KUKA KRL program: MyProgram_334().src

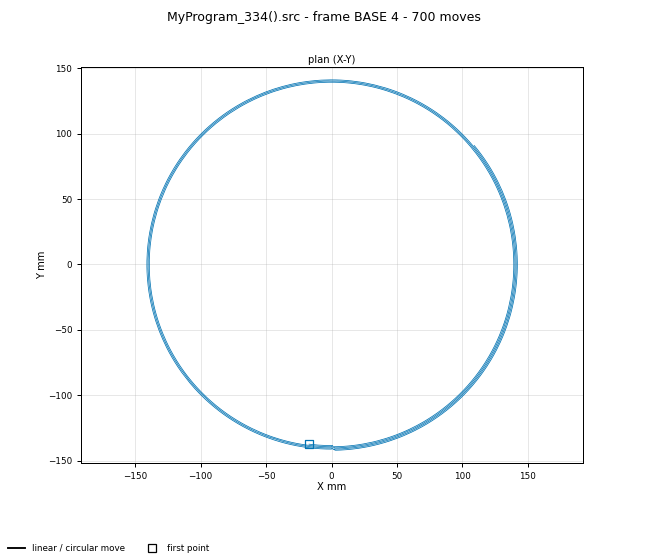
[picture p0: tool path of MyProgram_334().src in frame BASE 4, 700 of 700 moves have a stored position in this frame; points joined in program order, loops and branches not executed]
&ACCESS RVP
&REL 1
&PARAM TEMPLATE = C:\KRC\Roboter\Template\vorgabe
&PARAM EDITMASK = *
DEF MyProgram_334()
; ---- Setting reference (Base) ----
$BASE = BASE_DATA[4]

; --------------------------
; ---- Setting tool (TCP) ----
$TOOL = TOOL_DATA[3]
; --------------------------

$VEL.CP = VEL_APROX_PRINT
Startdeposition()
$VEL.CP = VEL_PRINT
LIN {X -17.1931,Y -137.3704,Z 189,A -88.3722,B 1.6874,C 0.25,E1 1.6941,E2 181.411} C_DIS
LIN {X -13.4645,Y -137.7837,Z 189,A -87.0235,B 1.6872,C 0.2509,E1 1.6978,E2 180.0902} C_DIS
LIN {X -10.3539,Y -138.0524,Z 189,A -85.5339,B 1.6873,C 0.25,E1 1.7021,E2 178.5723} C_DIS
LIN {X -7.0478,Y -138.2604,Z 189,A -84.1441,B 1.6873,C 0.2498,E1 1.706,E2 177.1792} C_DIS
LIN {X -4.0759,Y -138.3801,Z 189,A -82.9485,B 1.6873,C 0.2498,E1 1.7093,E2 175.9881} C_DIS
LIN {X 0.9672,Y -138.4367,Z 189,A -81.2262,B 1.6873,C 0.2508,E1 1.714,E2 174.316} C_DIS
Enddeposition()
LIN {X 0.9672,Y -138.4367,Z 189,A -81.2263,B 1.6873,C 0.2508,E1 1.714,E2 174.3161} C_DIS
Startdeposition()
$VEL.CP = VEL_PRINT
LIN {X -0.0441,Y -139.341,Z 189,A -81.8899,B 1.6847,C 0.2528,E1 1.7097,E2 175.0438} C_DIS
LIN {X -3.7886,Y -139.2876,Z 189,A -83.3825,B 1.6847,C 0.2528,E1 1.7056,E2 176.5304} C_DIS
LIN {X -7.5558,Y -139.1352,Z 189,A -85.0398,B 1.6846,C 0.2536,E1 1.7009,E2 178.2035} C_DIS
LIN {X -11.7168,Y -138.8455,Z 189,A -86.6706,B 1.6846,C 0.2533,E1 1.6963,E2 179.8232} C_DIS
LIN {X -16.1621,Y -138.3989,Z 189,A -88.4985,B 1.6846,C 0.2533,E1 1.6912,E2 181.6505} C_DIS
LIN {X -19.8344,Y -137.9201,Z 189,A -89.9991,B 1.6846,C 0.253,E1 1.6871,E2 183.1486} C_DIS
LIN {X -23.5368,Y -137.338,Z 189,A -91.6699,B 1.6846,C 0.2532,E1 1.6824,E2 184.8383} C_DIS
LIN {X -27.0838,Y -136.6831,Z 189,A -93.1243,B 1.6847,C 0.2527,E1 1.6784,E2 186.2892} C_DIS
LIN {X -30.8901,Y -135.8717,Z 189,A -95.0459,B 1.6847,C 0.2534,E1 1.673,E2 188.2563} C_DIS
LIN {X -34.6686,Y -134.9575,Z 189,A -96.3463,B 1.6849,C 0.2516,E1 1.6696,E2 189.5156} C_DIS
LIN {X -39.0122,Y -133.766,Z 189,A -97.892,B 1.6852,C 0.2496,E1 1.6655,E2 191.0188} C_DIS
LIN {X -44.1937,Y -132.1447,Z 189,A -100.3939,B 1.6852,C 0.2493,E1 1.6588,E2 193.5593} C_DIS
LIN {X -47.06,Y -131.1513,Z 189,A -101.7463,B 1.6852,C 0.2488,E1 1.6551,E2 194.9267} C_DIS
LIN {X -50.4559,Y -129.8824,Z 189,A -103.3021,B 1.6854,C 0.2479,E1 1.651,E2 196.492} C_DIS
LIN {X -54.7043,Y -128.1526,Z 189,A -105.2487,B 1.6856,C 0.2465,E1 1.646,E2 198.4475} C_DIS
LIN {X -58.2398,Y -126.5837,Z 189,A -106.757,B 1.6859,C 0.2448,E1 1.6421,E2 199.9446} C_DIS
LIN {X -61.123,Y -125.2179,Z 189,A -108.2374,B 1.6859,C 0.244,E1 1.6384,E2 201.4488} C_DIS
LIN {X -65.2655,Y -123.1094,Z 189,A -110.1627,B 1.6863,C 0.2421,E1 1.6336,E2 203.3763} C_DIS
LIN {X -69.2509,Y -120.9139,Z 189,A -112.1542,B 1.6865,C 0.2403,E1 1.6286,E2 205.3849} C_DIS
LIN {X -73.1981,Y -118.5664,Z 189,A -114.1264,B 1.6868,C 0.2382,E1 1.6239,E2 207.3689} C_DIS
LIN {X -76.997,Y -116.1355,Z 189,A -116.0185,B 1.6871,C 0.2358,E1 1.6194,E2 209.2664} C_DIS
LIN {X -80.6521,Y -113.6275,Z 189,A -117.9882,B 1.6875,C 0.2337,E1 1.6149,E2 211.2565} C_DIS
LIN {X -84.5138,Y -110.7846,Z 189,A -120.0169,B 1.6878,C 0.2309,E1 1.6103,E2 213.2931} C_DIS
LIN {X -88.1059,Y -107.9497,Z 189,A -121.9771,B 1.6882,C 0.2281,E1 1.606,E2 215.2641} C_DIS
LIN {X -91.9941,Y -104.6567,Z 189,A -124.2091,B 1.6886,C 0.225,E1 1.6012,E2 217.515} C_DIS
LIN {X -95.2914,Y -101.6638,Z 189,A -125.9306,B 1.6891,C 0.2216,E1 1.5977,E2 219.2212} C_DIS
LIN {X -99.9376,Y -97.0996,Z 189,A -128.9795,B 1.6896,C 0.2175,E1 1.5915,E2 222.321} C_DIS
LIN {X -103.139,Y -93.6917,Z 189,A -130.9753,B 1.6901,C 0.2139,E1 1.5877,E2 224.3266} C_DIS
LIN {X -105.5654,Y -90.949,Z 189,A -132.5877,B 1.6904,C 0.2112,E1 1.5847,E2 225.9533} C_DIS
LIN {X -108.5634,Y -87.3487,Z 189,A -134.6374,B 1.6909,C 0.2074,E1 1.5811,E2 228.0195} C_DIS
LIN {X -110.6317,Y -84.7137,Z 189,A -136.5253,B 1.6911,C 0.2054,E1 1.5778,E2 229.9766} C_DIS
LIN {X -113.2252,Y -81.215,Z 189,A -138.0383,B 1.6916,C 0.2011,E1 1.5753,E2 231.4516} C_DIS
LIN {X -115.7722,Y -77.5411,Z 189,A -140.0064,B 1.6921,C 0.1972,E1 1.5722,E2 233.4369} C_DIS
LIN {X -118.2406,Y -73.7223,Z 189,A -142.0402,B 1.6926,C 0.1932,E1 1.5691,E2 235.4924} C_DIS
LIN {X -120.7569,Y -69.5246,Z 189,A -144.164,B 1.6931,C 0.1887,E1 1.5661,E2 237.6307} C_DIS
LIN {X -122.8295,Y -65.7931,Z 189,A -146.1181,B 1.6935,C 0.1848,E1 1.5634,E2 239.611} C_DIS
LIN {X -124.8197,Y -61.9304,Z 189,A -147.9014,B 1.694,C 0.1804,E1 1.5612,E2 241.3932} C_DIS
LIN {X -126.4146,Y -58.6054,Z 189,A -149.3931,B 1.6944,C 0.1767,E1 1.5594,E2 242.881} C_DIS
LIN {X -127.825,Y -55.4619,Z 189,A -150.906,B 1.6947,C 0.1732,E1 1.5577,E2 244.4063} C_DIS
LIN {X -129.1309,Y -52.35,Z 189,A -152.5141,B 1.6951,C 0.17,E1 1.5559,E2 246.0435} C_DIS
LIN {X -130.4252,Y -49.0363,Z 189,A -154.5969,B 1.6954,C 0.1669,E1 1.5538,E2 248.2082} C_DIS
LIN {X -131.7948,Y -45.228,Z 189,A -156.3445,B 1.6958,C 0.1626,E1 1.5522,E2 249.9662} C_DIS
LIN {X -132.994,Y -41.5759,Z 189,A -157.7943,B 1.6962,C 0.1583,E1 1.551,E2 251.3981} C_DIS
LIN {X -134.1396,Y -37.7079,Z 189,A -159.4909,B 1.6966,C 0.1539,E1 1.5496,E2 253.0989} C_DIS
LIN {X -135.0311,Y -34.3786,Z 189,A -161.0191,B 1.6969,C 0.1502,E1 1.5486,E2 254.6411} C_DIS
LIN {X -135.8816,Y -30.8468,Z 189,A -162.6562,B 1.6973,C 0.1463,E1 1.5475,E2 256.2964} C_DIS
LIN {X -136.7225,Y -26.8848,Z 189,A -164.4513,B 1.6976,C 0.1419,E1 1.5465,E2 258.1078} C_DIS
LIN {X -137.3021,Y -23.7508,Z 189,A -165.9765,B 1.6979,C 0.1384,E1 1.5457,E2 259.6606} C_DIS
LIN {X -138.0556,Y -18.8842,Z 189,A -168.2312,B 1.6983,C 0.133,E1 1.5448,E2 261.9443} C_DIS
LIN {X -138.543,Y -14.872,Z 189,A -169.8988,B 1.6987,C 0.1284,E1 1.5443,E2 263.6116} C_DIS
LIN {X -138.8485,Y -11.6815,Z 189,A -171.525,B 1.699,C 0.125,E1 1.5439,E2 265.2772} C_DIS
LIN {X -139.266,Y -4.5657,Z 189,A -174.6514,B 1.6995,C 0.1169,E1 1.5434,E2 268.4273} C_DIS
LIN {X -139.2951,Y 3.5199,Z 189,A -178.0329,B 1.7001,C 0.1077,E1 1.5434,E2 271.8141} C_DIS
LIN {X -138.9355,Y 10.6065,Z 189,A 178.5798,B 1.7006,C 0.0998,E1 1.544,E2 275.2602} C_DIS
LIN {X -138.6283,Y 14.0762,Z 189,A 176.1293,B 1.7008,C 0.0965,E1 1.5448,E2 277.8391} C_DIS
LIN {X -137.8333,Y 20.4416,Z 189,A 173.9114,B 1.7012,C 0.0889,E1 1.5456,E2 280.0024} C_DIS
LIN {X -136.9608,Y 25.6386,Z 189,A 171.7478,B 1.7015,C 0.0829,E1 1.5466,E2 282.1642} C_DIS
LIN {X -136.3322,Y 28.7963,Z 189,A 170.4206,B 1.7017,C 0.0793,E1 1.5474,E2 283.4909} C_DIS
LIN {X -135.3028,Y 33.3,Z 189,A 168.3355,B 1.7019,C 0.0743,E1 1.5487,E2 285.5982} C_DIS
LIN {X -134.2479,Y 37.3205,Z 189,A 166.4669,B 1.7021,C 0.0698,E1 1.5501,E2 287.4856} C_DIS
LIN {X -133.354,Y 40.3998,Z 189,A 164.9943,B 1.7023,C 0.0664,E1 1.5513,E2 288.9767} C_DIS
LIN {X -132.2704,Y 43.8161,Z 189,A 163.3966,B 1.7023,C 0.0626,E1 1.5526,E2 290.5889} C_DIS
LIN {X -130.1769,Y 49.6984,Z 189,A 159.3255,B 1.7026,C 0.0571,E1 1.5568,E2 294.8438} C_DIS
LIN {X -127.0258,Y 57.2699,Z 189,A 156.9836,B 1.7029,C 0.0477,E1 1.5593,E2 297.0569} C_DIS
LIN {X -125.792,Y 59.9301,Z 189,A 155.5142,B 1.7029,C 0.0449,E1 1.5611,E2 298.558} C_DIS
LIN {X -123.5927,Y 64.3452,Z 189,A 153.4761,B 1.7031,C 0.04,E1 1.5637,E2 300.596} C_DIS
LIN {X -121.6059,Y 68.0285,Z 189,A 151.5327,B 1.7031,C 0.0361,E1 1.5663,E2 302.5657} C_DIS
LIN {X -118.915,Y 72.6297,Z 189,A 149.1411,B 1.7033,C 0.0312,E1 1.5698,E2 304.9802} C_DIS
LIN {X -116.5349,Y 76.3903,Z 189,A 147.1766,B 1.7033,C 0.0271,E1 1.5728,E2 306.9598} C_DIS
LIN {X -114.0033,Y 80.1192,Z 189,A 144.3261,B 1.7033,C 0.0242,E1 1.5776,E2 309.9294} C_DIS
LIN {X -109.9869,Y 85.5495,Z 189,A 142.2547,B 1.7035,C 0.0174,E1 1.5809,E2 311.914} C_DIS
LIN {X -107.2118,Y 89.0025,Z 189,A 140.3124,B 1.7035,C 0.0138,E1 1.5844,E2 313.8697} C_DIS
LIN {X -104.2149,Y 92.4938,Z 189,A 138.3109,B 1.7035,C 0.0101,E1 1.5881,E2 315.8831} C_DIS
LIN {X -101.2783,Y 95.7001,Z 189,A 136.4166,B 1.7035,C 0.0068,E1 1.5917,E2 317.789} C_DIS
LIN {X -98.0861,Y 98.9694,Z 189,A 134.44,B 1.7035,C 0.0035,E1 1.5956,E2 319.776} C_DIS
LIN {X -94.9208,Y 102.009,Z 189,A 132.5493,B 1.7035,C 0.0004,E1 1.5995,E2 321.6759} C_DIS
LIN {X -91.854,Y 104.7794,Z 189,A 130.6632,B 1.7035,C -0.0022,E1 1.6035,E2 323.5832} C_DIS
LIN {X -88.2502,Y 107.8318,Z 189,A 128.6575,B 1.7035,C -0.0053,E1 1.6078,E2 325.5952} C_DIS
LIN {X -84.6059,Y 110.7142,Z 189,A 126.6699,B 1.7035,C -0.0081,E1 1.6122,E2 327.5907} C_DIS
LIN {X -82.3482,Y 112.4037,Z 189,A 124.8215,B 1.7035,C -0.0085,E1 1.6166,E2 329.5199} C_DIS
LIN {X -77.8924,Y 115.5363,Z 189,A 123.0914,B 1.7035,C -0.0127,E1 1.6205,E2 331.1884} C_DIS
LIN {X -70.8213,Y 120.0009,Z 189,A 119.2961,B 1.7035,C -0.0164,E1 1.6296,E2 335.0238} C_DIS
LIN {X -67.8418,Y 121.7104,Z 189,A 118.0665,B 1.7035,C -0.0184,E1 1.6326,E2 336.2309} C_DIS
LIN {X -63.7531,Y 123.8996,Z 189,A 116.1252,B 1.7035,C -0.0204,E1 1.6374,E2 338.1751} C_DIS
LIN {X -59.0879,Y 126.1915,Z 189,A 113.862,B 1.7035,C -0.0223,E1 1.6431,E2 340.4519} C_DIS
LIN {X -56.22,Y 127.4954,Z 189,A 112.1277,B 1.7035,C -0.0223,E1 1.6477,E2 342.237} C_DIS
LIN {X -52.2271,Y 129.1804,Z 189,A 110.8298,B 1.7034,C -0.0251,E1 1.6509,E2 343.4769} C_DIS
LIN {X -49.1078,Y 130.3984,Z 189,A 109.4562,B 1.7034,C -0.0262,E1 1.6545,E2 344.8494} C_DIS
LIN {X -46.1666,Y 131.4694,Z 189,A 108.0229,B 1.7034,C -0.0267,E1 1.6583,E2 346.2993} C_DIS
LIN {X -43.1974,Y 132.4762,Z 189,A 106.6318,B 1.7034,C -0.0273,E1 1.6621,E2 347.7017} C_DIS
LIN {X -39.4643,Y 133.6336,Z 189,A 105.1838,B 1.7034,C -0.0287,E1 1.6659,E2 349.1301} C_DIS
LIN {X -36.6681,Y 134.4298,Z 189,A 103.8373,B 1.7034,C -0.0288,E1 1.6696,E2 350.4938} C_DIS
LIN {X -33.0265,Y 135.3687,Z 189,A 102.418,B 1.7033,C -0.0299,E1 1.6734,E2 351.8972} C_DIS
LIN {X -26.5552,Y 136.7856,Z 189,A 99.7769,B 1.7033,C -0.0311,E1 1.6806,E2 354.5272} C_DIS
LIN {X -20.2885,Y 137.8552,Z 189,A 96.8986,B 1.7033,C -0.0308,E1 1.6887,E2 357.4355} C_DIS
LIN {X -13.7379,Y 138.6607,Z 189,A 94.2177,B 1.7033,C -0.0311,E1 1.6961,E2 360.1113} C_DIS
LIN {X -10.405,Y 138.9502,Z 189,A 92.8469,B 1.7033,C -0.0311,E1 1.7,E2 361.4809} C_DIS
LIN {X -6.6749,Y 139.1795,Z 189,A 91.2384,B 1.7033,C -0.0307,E1 1.7045,E2 363.0973} C_DIS
LIN {X -2.3484,Y 139.3193,Z 189,A 89.508,B 1.7033,C -0.0305,E1 1.7093,E2 364.8211} C_DIS
LIN {X 2.1061,Y 139.3234,Z 189,A 87.7266,B 1.7033,C -0.0302,E1 1.7143,E2 366.5958} C_DIS
LIN {X 5.8309,Y 139.2176,Z 189,A 86.1325,B 1.7033,C -0.0295,E1 1.7188,E2 368.1966} C_DIS
LIN {X 9.9521,Y 138.9833,Z 189,A 84.5416,B 1.7033,C -0.0292,E1 1.7232,E2 369.7743} C_DIS
LIN {X 13.9658,Y 138.6389,Z 189,A 82.8076,B 1.7033,C -0.028,E1 1.7281,E2 371.5169} C_DIS
LIN {X 18.0492,Y 138.165,Z 189,A 81.2711,B 1.7033,C -0.0277,E1 1.7323,E2 373.0347} C_DIS
LIN {X 22.3782,Y 137.5313,Z 189,A 79.2427,B 1.7033,C -0.0255,E1 1.738,E2 375.0896} C_DIS
LIN {X 25.5538,Y 136.977,Z 189,A 78.298,B 1.7033,C -0.0261,E1 1.7405,E2 375.989} C_DIS
LIN {X 30.7367,Y 135.9067,Z 189,A 76.074,B 1.7033,C -0.0241,E1 1.7466,E2 378.218} C_DIS
LIN {X 34.1296,Y 135.0943,Z 189,A 74.6963,B 1.7033,C -0.0231,E1 1.7503,E2 379.5886} C_DIS
LIN {X 37.6281,Y 134.1619,Z 189,A 72.7762,B 1.7034,C -0.0197,E1 1.7556,E2 381.5593} C_DIS
LIN {X 41.8649,Y 132.9019,Z 189,A 71.4394,B 1.7034,C -0.02,E1 1.7591,E2 382.839} C_DIS
LIN {X 45.3787,Y 131.7426,Z 189,A 70.0078,B 1.7034,C -0.0188,E1 1.7628,E2 384.2596} C_DIS
LIN {X 48.496,Y 130.6275,Z 189,A 68.5927,B 1.7034,C -0.0169,E1 1.7666,E2 385.6808} C_DIS
LIN {X 52.2217,Y 129.1826,Z 189,A 67.1299,B 1.7034,C -0.0157,E1 1.7703,E2 387.1218} C_DIS
LIN {X 55.2285,Y 127.926,Z 189,A 65.8364,B 1.7034,C -0.0142,E1 1.7736,E2 388.4096} C_DIS
LIN {X 59.0595,Y 126.2046,Z 189,A 64.2665,B 1.7035,C -0.0127,E1 1.7776,E2 389.9604} C_DIS
LIN {X 63.2117,Y 124.1753,Z 189,A 62.3533,B 1.7035,C -0.0099,E1 1.7824,E2 391.8749} C_DIS
LIN {X 66.4287,Y 122.4873,Z 189,A 60.8272,B 1.7035,C -0.0075,E1 1.7862,E2 393.4049} C_DIS
LIN {X 70.2667,Y 120.3267,Z 189,A 59.0504,B 1.7035,C -0.0048,E1 1.7905,E2 395.1773} C_DIS
LIN {X 74.2047,Y 117.9385,Z 189,A 57.3258,B 1.7035,C -0.0026,E1 1.7946,E2 396.8815} C_DIS
LIN {X 77.6638,Y 115.6903,Z 189,A 55.6731,B 1.7035,C 0.0001,E1 1.7984,E2 398.5289} C_DIS
LIN {X 81.7267,Y 112.8563,Z 189,A 53.7387,B 1.7035,C 0.0031,E1 1.8028,E2 400.4509} C_DIS
LIN {X 85.4168,Y 110.0898,Z 189,A 51.9673,B 1.7035,C 0.0059,E1 1.8067,E2 402.2073} C_DIS
LIN {X 88.472,Y 107.6505,Z 189,A 50.3371,B 1.7035,C 0.0091,E1 1.8103,E2 403.8403} C_DIS
LIN {X 91.8975,Y 104.7412,Z 189,A 47.6672,B 1.7035,C 0.0176,E1 1.8161,E2 406.609} C_DIS
LIN {X 97.8168,Y 99.236,Z 189,A 45.5288,B 1.7035,C 0.0175,E1 1.8201,E2 408.6048} C_DIS
LIN {X 101.022,Y 95.9715,Z 189,A 43.7434,B 1.7035,C 0.0209,E1 1.8235,E2 410.3788} C_DIS
LIN {X 103.6866,Y 93.0855,Z 189,A 42.1654,B 1.7034,C 0.0242,E1 1.8265,E2 411.9524} C_DIS
LIN {X 106.0523,Y 90.381,Z 189,A 40.0198,B 1.7033,C 0.0316,E1 1.8306,E2 414.1796} C_DIS
LIN {X 110.5834,Y 84.7768,Z 189,A 38.0771,B 1.7033,C 0.0321,E1 1.8337,E2 415.9984} C_DIS
LIN {X 113.2671,Y 81.1564,Z 189,A 36.3543,B 1.7032,C 0.0356,E1 1.8365,E2 417.7055} C_DIS
LIN {X 115.9379,Y 77.2929,Z 189,A 34.7596,B 1.7032,C 0.0381,E1 1.8389,E2 419.2589} C_DIS
LIN {X 118.1227,Y 73.9116,Z 189,A 32.9931,B 1.703,C 0.0428,E1 1.8416,E2 421.0396} C_DIS
LIN {X 120.467,Y 70.0253,Z 189,A 31.2769,B 1.703,C 0.0464,E1 1.844,E2 422.7376} C_DIS
LIN {X 122.6319,Y 66.161,Z 189,A 29.5644,B 1.7028,C 0.0503,E1 1.8463,E2 424.4371} C_DIS
LIN {X 124.7052,Y 62.1625,Z 189,A 27.7886,B 1.7027,C 0.0545,E1 1.8485,E2 426.2039} C_DIS
LIN {X 126.4151,Y 58.6043,Z 189,A 26.0578,B 1.7025,C 0.0594,E1 1.8506,E2 427.9487} C_DIS
LIN {X 128.0393,Y 54.9665,Z 189,A 24.8738,B 1.7025,C 0.0607,E1 1.8519,E2 429.0763} C_DIS
LIN {X 129.6816,Y 50.9726,Z 189,A 23.2034,B 1.7023,C 0.0646,E1 1.8536,E2 430.7341} C_DIS
LIN {X 130.946,Y 47.6293,Z 189,A 21.87,B 1.7023,C 0.0676,E1 1.8549,E2 432.0508} C_DIS
LIN {X 132.1097,Y 44.2987,Z 189,A 20.5344,B 1.7021,C 0.0707,E1 1.856,E2 433.3724} C_DIS
LIN {X 133.1818,Y 40.9624,Z 189,A 19.3184,B 1.702,C 0.0731,E1 1.857,E2 434.5604} C_DIS
LIN {X 134.1223,Y 37.7696,Z 189,A 17.8219,B 1.7018,C 0.0777,E1 1.8582,E2 436.0738} C_DIS
LIN {X 135.386,Y 32.9546,Z 189,A 16.0354,B 1.7016,C 0.0815,E1 1.8594,E2 437.8279} C_DIS
LIN {X 136.0407,Y 30.1465,Z 189,A 14.6824,B 1.7014,C 0.0859,E1 1.8603,E2 439.203} C_DIS
LIN {X 136.7328,Y 26.8313,Z 189,A 12.9859,B 1.7011,C 0.0918,E1 1.8612,E2 440.9388} C_DIS
LIN {X 137.7291,Y 21.1203,Z 189,A 11.4647,B 1.7011,C 0.0925,E1 1.8618,E2 442.351} C_DIS
LIN {X 138.3117,Y 16.8926,Z 189,A 9.8044,B 1.7008,C 0.0967,E1 1.8624,E2 444} C_DIS
LIN {X 138.757,Y 12.735,Z 189,A 8.1992,B 1.7006,C 0.1007,E1 1.8628,E2 445.5914} C_DIS
LIN {X 139.0681,Y 8.6863,Z 189,A 6.6628,B 1.7003,C 0.1044,E1 1.8631,E2 447.1115} C_DIS
LIN {X 139.2773,Y 4.1607,Z 189,A 4.9626,B 1.7001,C 0.1085,E1 1.8633,E2 448.7916} C_DIS
LIN {X 139.3426,Y -0.0212,Z 189,A 3.2601,B 1.6998,C 0.1132,E1 1.8633,E2 450.4929} C_DIS
LIN {X 139.2828,Y -3.9625,Z 189,A 1.8826,B 1.6996,C 0.1161,E1 1.8633,E2 451.8395} C_DIS
LIN {X 139.0921,Y -8.2964,Z 189,A 0.2588,B 1.6993,C 0.1199,E1 1.863,E2 453.4435} C_DIS
LIN {X 138.8503,Y -11.6602,Z 189,A -1.0357,B 1.6991,C 0.1232,E1 1.8628,E2 454.7268} C_DIS
LIN {X 138.451,Y -15.7255,Z 189,A -2.7113,B 1.6987,C 0.1278,E1 1.8623,E2 456.403} C_DIS
LIN {X 137.9225,Y -19.817,Z 189,A -4.118,B 1.6985,C 0.1305,E1 1.8618,E2 457.7726} C_DIS
LIN {X 137.2685,Y -23.9387,Z 189,A -5.796,B 1.6982,C 0.135,E1 1.861,E2 459.4467} C_DIS
LIN {X 135.2979,Y -33.319,Z 189,A -9.5804,B 1.6974,C 0.1448,E1 1.8587,E2 463.2131} C_DIS
LIN {X 134.1247,Y -37.7611,Z 189,A -11.1161,B 1.6972,C 0.1474,E1 1.8576,E2 464.7031} C_DIS
LIN {X 133.1318,Y -41.1259,Z 189,A -12.4778,B 1.6969,C 0.1508,E1 1.8566,E2 466.055} C_DIS
LIN {X 131.9622,Y -44.7416,Z 189,A -14.0163,B 1.6965,C 0.1548,E1 1.8552,E2 467.5915} C_DIS
LIN {X 130.5757,Y -48.6342,Z 189,A -15.4923,B 1.6962,C 0.1578,E1 1.8538,E2 469.0388} C_DIS
LIN {X 129.3898,Y -51.7078,Z 189,A -16.7612,B 1.696,C 0.1607,E1 1.8525,E2 470.2972} C_DIS
LIN {X 128.1526,Y -54.7043,Z 189,A -18.0545,B 1.6956,C 0.164,E1 1.8511,E2 471.5862} C_DIS
LIN {X 126.5706,Y -58.268,Z 189,A -19.8906,B 1.6951,C 0.1697,E1 1.849,E2 473.4546} C_DIS
LIN {X 124.6622,Y -62.2496,Z 189,A -21.1859,B 1.695,C 0.1708,E1 1.8474,E2 474.6815} C_DIS
LIN {X 122.6916,Y -66.0498,Z 189,A -22.8434,B 1.6946,C 0.1746,E1 1.8453,E2 476.3264} C_DIS
LIN {X 120.4835,Y -69.9969,Z 189,A -24.3703,B 1.6943,C 0.1769,E1 1.8433,E2 477.8096} C_DIS
LIN {X 117.5522,Y -74.8158,Z 189,A -26.783,B 1.6937,C 0.1833,E1 1.8397,E2 480.2369} C_DIS
LIN {X 115.1007,Y -78.5351,Z 189,A -28.4661,B 1.6933,C 0.1867,E1 1.8371,E2 481.9011} C_DIS
LIN {X 112.5772,Y -82.1117,Z 189,A -30.1714,B 1.6929,C 0.1903,E1 1.8343,E2 483.5949} C_DIS
LIN {X 109.8894,Y -85.6753,Z 189,A -31.8934,B 1.6925,C 0.1938,E1 1.8314,E2 485.3029} C_DIS
LIN {X 107.0457,Y -89.2031,Z 189,A -33.6546,B 1.6921,C 0.1973,E1 1.8283,E2 487.0516} C_DIS
LIN {X 104.0361,Y -92.6952,Z 189,A -35.3941,B 1.6917,C 0.2005,E1 1.8252,E2 488.7712} C_DIS
LIN {X 101.0402,Y -95.9524,Z 189,A -37.1387,B 1.6913,C 0.204,E1 1.8219,E2 490.5069} C_DIS
LIN {X 97.8572,Y -99.1964,Z 189,A -38.8934,B 1.6909,C 0.2072,E1 1.8184,E2 492.2474} C_DIS
LIN {X 94.7241,Y -102.1921,Z 189,A -40.5265,B 1.6906,C 0.2099,E1 1.8151,E2 493.8613} C_DIS
LIN {X 91.4289,Y -105.1503,Z 189,A -42.2488,B 1.6902,C 0.2129,E1 1.8115,E2 495.5714} C_DIS
LIN {X 87.9437,Y -108.0823,Z 189,A -44.0306,B 1.6898,C 0.2159,E1 1.8077,E2 497.3421} C_DIS
LIN {X 84.4557,Y -110.8291,Z 189,A -45.7473,B 1.6895,C 0.2187,E1 1.804,E2 499.045} C_DIS
LIN {X 80.8237,Y -113.505,Z 189,A -47.5114,B 1.6891,C 0.2215,E1 1.8,E2 500.798} C_DIS
LIN {X 77.099,Y -116.0674,Z 189,A -49.307,B 1.6887,C 0.2243,E1 1.7958,E2 502.5861} C_DIS
LIN {X 73.2339,Y -118.5444,Z 189,A -51.1295,B 1.6883,C 0.2271,E1 1.7915,E2 504.401} C_DIS
LIN {X 69.8132,Y -120.5898,Z 189,A -52.786,B 1.688,C 0.2299,E1 1.7875,E2 506.0611} C_DIS
LIN {X 65.2742,Y -123.1049,Z 189,A -54.6664,B 1.6877,C 0.2316,E1 1.783,E2 507.9079} C_DIS
LIN {X 61.758,Y -124.9047,Z 189,A -56.0919,B 1.6876,C 0.2329,E1 1.7795,E2 509.3068} C_DIS
LIN {X 59.5818,Y -125.9584,Z 189,A -57.4739,B 1.6871,C 0.2365,E1 1.7759,E2 510.7435} C_DIS
LIN {X 56.0716,Y -127.5614,Z 189,A -58.721,B 1.6871,C 0.2367,E1 1.7728,E2 511.9446} C_DIS
LIN {X 52.5479,Y -129.0511,Z 189,A -60.1847,B 1.6868,C 0.2382,E1 1.769,E2 513.3939} C_DIS
LIN {X 49.1274,Y -130.391,Z 189,A -61.6234,B 1.6866,C 0.2396,E1 1.7653,E2 514.8236} C_DIS
LIN {X 45.889,Y -131.5657,Z 189,A -63.0155,B 1.6864,C 0.2411,E1 1.7616,E2 516.2133} C_DIS
LIN {X 41.297,Y -133.0794,Z 189,A -64.9301,B 1.6861,C 0.2429,E1 1.7565,E2 518.119} C_DIS
LIN {X 37.8758,Y -134.0926,Z 189,A -66.2334,B 1.6861,C 0.2436,E1 1.7531,E2 519.4002} C_DIS
LIN {X 34.7127,Y -134.9464,Z 189,A -67.5959,B 1.6859,C 0.245,E1 1.7494,E2 520.7657} C_DIS
LIN {X 31.1527,Y -135.8117,Z 189,A -69.0989,B 1.6857,C 0.2463,E1 1.7453,E2 522.2691} C_DIS
LIN {X 24.2419,Y -137.2142,Z 189,A -72.0306,B 1.6853,C 0.2488,E1 1.7372,E2 525.2071} C_DIS
LIN {X 19.9077,Y -137.9096,Z 189,A -73.7516,B 1.6852,C 0.2496,E1 1.7325,E2 526.9173} C_DIS
LIN {X 16.1923,Y -138.3953,Z 189,A -75.2874,B 1.685,C 0.2505,E1 1.7282,E2 528.4534} C_DIS
LIN {X 12.2007,Y -138.8046,Z 189,A -76.9205,B 1.685,C 0.2513,E1 1.7236,E2 530.0851} C_DIS
LIN {X 8.3564,Y -139.0884,Z 189,A -78.4915,B 1.6848,C 0.252,E1 1.7192,E2 531.6549} C_DIS
LIN {X 4.276,Y -139.2741,Z 189,A -80.1327,B 1.6848,C 0.2524,E1 1.7146,E2 533.2916} C_DIS
LIN {X 0.9753,Y -139.3318,Z 189,A -81.0158,B 1.685,C 0.2507,E1 1.7124,E2 534.1083} C_DIS
Enddeposition()
LIN {X 0.9753,Y -139.3318,Z 189,A -81.0159,B 1.685,C 0.2507,E1 1.7124,E2 534.1085} C_DIS
Startdeposition()
$VEL.CP = VEL_PRINT
LIN {X 2.4357,Y -140.2172,Z 189,A -80.1883,B 1.6828,C 0.2502,E1 1.7124,E2 533.2763} C_DIS
LIN {X 5.5567,Y -140.1281,Z 189,A -78.9013,B 1.6828,C 0.2497,E1 1.716,E2 531.9871} C_DIS
LIN {X 9.913,Y -139.8877,Z 189,A -77.1417,B 1.683,C 0.249,E1 1.721,E2 530.2299} C_DIS
LIN {X 13.4287,Y -139.5937,Z 189,A -75.7327,B 1.683,C 0.2484,E1 1.7249,E2 528.8247} C_DIS
LIN {X 17.6824,Y -139.1199,Z 189,A -73.9611,B 1.6832,C 0.2472,E1 1.7298,E2 527.0488} C_DIS
LIN {X 21.4972,Y -138.5806,Z 189,A -72.5062,B 1.6833,C 0.2468,E1 1.7338,E2 525.61} C_DIS
LIN {X 24.5585,Y -138.071,Z 189,A -70.9548,B 1.6837,C 0.2444,E1 1.7382,E2 524.0173} C_DIS
LIN {X 27.9106,Y -137.4325,Z 189,A -69.5808,B 1.6838,C 0.2434,E1 1.742,E2 522.6453} C_DIS
LIN {X 31.3254,Y -136.6946,Z 189,A -68.4769,B 1.6838,C 0.2438,E1 1.7449,E2 521.5868} C_DIS
LIN {X 34.7623,Y -135.8614,Z 189,A -67.1298,B 1.6838,C 0.243,E1 1.7485,E2 520.2528} C_DIS
LIN {X 38.0974,Y -134.9643,Z 189,A -65.7051,B 1.6841,C 0.2415,E1 1.7524,E2 518.8252} C_DIS
LIN {X 43.694,Y -133.2587,Z 189,A -63.4775,B 1.6843,C 0.2398,E1 1.7583,E2 516.6193} C_DIS
LIN {X 47.7876,Y -131.8447,Z 189,A -61.734,B 1.6846,C 0.2379,E1 1.7629,E2 514.8783} C_DIS
LIN {X 51.0066,Y -130.6331,Z 189,A -60.3457,B 1.6848,C 0.2363,E1 1.7665,E2 513.4914} C_DIS
LIN {X 54.0514,Y -129.4027,Z 189,A -59.0155,B 1.6851,C 0.2346,E1 1.77,E2 512.1619} C_DIS
LIN {X 62.2492,Y -125.665,Z 189,A -55.5627,B 1.6856,C 0.2308,E1 1.7787,E2 508.7392} C_DIS
LIN {X 64.9888,Y -124.2703,Z 189,A -53.721,B 1.6863,C 0.2255,E1 1.7834,E2 506.8132} C_DIS
LIN {X 69.6033,Y -121.748,Z 189,A -52.1642,B 1.6863,C 0.2257,E1 1.787,E2 505.3393} C_DIS
LIN {X 73.3265,Y -119.5424,Z 189,A -50.4657,B 1.6866,C 0.2232,E1 1.7911,E2 503.6493} C_DIS
LIN {X 77.3345,Y -116.9898,Z 189,A -48.6261,B 1.687,C 0.2205,E1 1.7954,E2 501.8226} C_DIS
LIN {X 81.1552,Y -114.3729,Z 189,A -46.8263,B 1.6873,C 0.2177,E1 1.7995,E2 500.0346} C_DIS
LIN {X 84.8295,Y -111.675,Z 189,A -45.0411,B 1.6877,C 0.2148,E1 1.8035,E2 498.2588} C_DIS
LIN {X 88.3555,Y -108.9065,Z 189,A -43.3156,B 1.6881,C 0.2119,E1 1.8072,E2 496.5469} C_DIS
LIN {X 91.8818,Y -105.9485,Z 189,A -41.5278,B 1.6884,C 0.2088,E1 1.811,E2 494.7707} C_DIS
LIN {X 95.2989,Y -102.8855,Z 189,A -39.757,B 1.6888,C 0.2057,E1 1.8146,E2 493.0131} C_DIS
LIN {X 98.5502,Y -99.7757,Z 189,A -38.0616,B 1.6892,C 0.2028,E1 1.818,E2 491.3363} C_DIS
LIN {X 101.5311,Y -96.7402,Z 189,A -36.4487,B 1.6895,C 0.1999,E1 1.8211,E2 489.7396} C_DIS
LIN {X 104.5416,Y -93.4785,Z 189,A -34.7229,B 1.6899,C 0.1965,E1 1.8243,E2 488.0246} C_DIS
LIN {X 107.5762,Y -89.9699,Z 189,A -32.936,B 1.6903,C 0.193,E1 1.8275,E2 486.2513} C_DIS
LIN {X 110.2593,Y -86.6606,Z 189,A -31.2957,B 1.6907,C 0.1897,E1 1.8304,E2 484.6238} C_DIS
LIN {X 113.0904,Y -82.9322,Z 189,A -29.5173,B 1.6911,C 0.1861,E1 1.8333,E2 482.8625} C_DIS
LIN {X 115.7819,Y -79.1315,Z 189,A -27.7342,B 1.6915,C 0.1824,E1 1.8361,E2 481.0946} C_DIS
LIN {X 118.3264,Y -75.2741,Z 189,A -25.7507,B 1.6921,C 0.1772,E1 1.8392,E2 479.0964} C_DIS
LIN {X 120.1997,Y -72.2444,Z 189,A -24.416,B 1.6923,C 0.1744,E1 1.8411,E2 477.7773} C_DIS
LIN {X 121.9467,Y -69.255,Z 189,A -23.3729,B 1.6924,C 0.1735,E1 1.8424,E2 476.7845} C_DIS
LIN {X 123.3348,Y -66.7525,Z 189,A -22.1798,B 1.6928,C 0.1703,E1 1.844,E2 475.5873} C_DIS
LIN {X 125.2426,Y -63.097,Z 189,A -20.5589,B 1.6931,C 0.1665,E1 1.8461,E2 473.9738} C_DIS
LIN {X 127.7761,Y -57.7946,Z 189,A -18.5893,B 1.6935,C 0.1633,E1 1.8484,E2 472.0618} C_DIS
LIN {X 129,Y -55.01,Z 189,A -17.3567,B 1.6938,C 0.1601,E1 1.8497,E2 470.8296} C_DIS
LIN {X 130.0577,Y -52.4558,Z 189,A -16.2697,B 1.694,C 0.1574,E1 1.8509,E2 469.7476} C_DIS
LIN {X 131.4796,Y -48.7846,Z 189,A -14.7366,B 1.6944,C 0.1537,E1 1.8524,E2 468.2237} C_DIS
LIN {X 133.528,Y -42.8597,Z 189,A -12.6502,B 1.6947,C 0.1502,E1 1.8542,E2 466.2} C_DIS
LIN {X 134.3033,Y -40.3703,Z 189,A -11.452,B 1.695,C 0.1464,E1 1.8552,E2 464.9831} C_DIS
LIN {X 135.3132,Y -36.8449,Z 189,A -9.4799,B 1.6956,C 0.1389,E1 1.8567,E2 462.9454} C_DIS
LIN {X 136.5835,Y -31.8119,Z 189,A -8.1808,B 1.6956,C 0.1389,E1 1.8575,E2 461.7565} C_DIS
LIN {X 137.238,Y -28.8615,Z 189,A -6.9666,B 1.6959,C 0.1357,E1 1.8582,E2 460.5443} C_DIS
LIN {X 137.8782,Y -25.6283,Z 189,A -5.6742,B 1.6961,C 0.1324,E1 1.8588,E2 459.2583} C_DIS
LIN {X 138.582,Y -21.4881,Z 189,A -4.1258,B 1.6964,C 0.1288,E1 1.8595,E2 457.7313} C_DIS
LIN {X 139.0771,Y -18.0094,Z 189,A -2.8174,B 1.6967,C 0.1257,E1 1.86,E2 456.439} C_DIS
LIN {X 139.4745,Y -14.6196,Z 189,A -1.4529,B 1.6969,C 0.122,E1 1.8604,E2 455.0777} C_DIS
LIN {X 139.8613,Y -10.2745,Z 189,A 0.1648,B 1.6972,C 0.1182,E1 1.8608,E2 453.4809} C_DIS
LIN {X 140.0889,Y -6.4926,Z 189,A 1.6846,B 1.6975,C 0.1141,E1 1.861,E2 451.9639} C_DIS
LIN {X 140.2184,Y -2.3584,Z 189,A 3.114,B 1.6977,C 0.1112,E1 1.8611,E2 450.5682} C_DIS
LIN {X 140.2352,Y 1.0569,Z 189,A 4.5505,B 1.6979,C 0.107,E1 1.8611,E2 449.1254} C_DIS
LIN {X 140.1209,Y 5.743,Z 189,A 6.2343,B 1.6982,C 0.1033,E1 1.8609,E2 447.4712} C_DIS
LIN {X 139.8792,Y 10.0301,Z 189,A 7.8239,B 1.6984,C 0.0995,E1 1.8607,E2 445.9024} C_DIS
LIN {X 139.569,Y 13.6858,Z 189,A 9.1693,B 1.6986,C 0.0964,E1 1.8603,E2 444.5764} C_DIS
LIN {X 139.1476,Y 17.4712,Z 189,A 10.67,B 1.6988,C 0.0925,E1 1.8598,E2 443.0823} C_DIS
LIN {X 138.5889,Y 21.4435,Z 189,A 12.2222,B 1.699,C 0.0885,E1 1.8592,E2 441.5405} C_DIS
LIN {X 137.7502,Y 26.2978,Z 189,A 13.7357,B 1.6991,C 0.0864,E1 1.8585,E2 440.0913} C_DIS
LIN {X 136.7661,Y 31.0124,Z 189,A 15.7478,B 1.6994,C 0.0807,E1 1.8574,E2 438.0727} C_DIS
LIN {X 136.2171,Y 33.3438,Z 189,A 16.7203,B 1.6995,C 0.0781,E1 1.8567,E2 437.1005} C_DIS
LIN {X 134.6912,Y 39.0522,Z 189,A 18.8056,B 1.6997,C 0.0738,E1 1.8552,E2 435.0568} C_DIS
LIN {X 133.4616,Y 43.0675,Z 189,A 20.5601,B 1.6999,C 0.0689,E1 1.8537,E2 433.2966} C_DIS
LIN {X 132.4208,Y 46.1674,Z 189,A 21.8115,B 1.7,C 0.0659,E1 1.8526,E2 432.0557} C_DIS
LIN {X 131.2131,Y 49.4962,Z 189,A 23.1237,B 1.7001,C 0.063,E1 1.8514,E2 430.7603} C_DIS
LIN {X 129.9335,Y 52.7641,Z 189,A 24.4782,B 1.7003,C 0.0597,E1 1.85,E2 429.4154} C_DIS
LIN {X 128.7745,Y 55.5317,Z 189,A 25.8048,B 1.7003,C 0.0558,E1 1.8485,E2 428.0754} C_DIS
LIN {X 126.7257,Y 60.0616,Z 189,A 27.35,B 1.7005,C 0.0538,E1 1.8468,E2 426.5919} C_DIS
LIN {X 125.0267,Y 63.5212,Z 189,A 28.9531,B 1.7005,C 0.0496,E1 1.8448,E2 424.9847} C_DIS
LIN {X 123.2961,Y 66.8236,Z 189,A 30.4959,B 1.7007,C 0.0457,E1 1.8427,E2 423.439} C_DIS
LIN {X 120.9755,Y 70.9375,Z 189,A 32.2599,B 1.7007,C 0.0419,E1 1.8403,E2 421.6956} C_DIS
LIN {X 118.5899,Y 74.8573,Z 189,A 34.4278,B 1.7009,C 0.0355,E1 1.837,E2 419.4898} C_DIS
LIN {X 115.9722,Y 78.8524,Z 189,A 35.5163,B 1.7009,C 0.0364,E1 1.8355,E2 418.5105} C_DIS
LIN {X 113.1381,Y 82.8672,Z 189,A 37.7203,B 1.701,C 0.0304,E1 1.8319,E2 416.2814} C_DIS
LIN {X 109.9951,Y 86.9949,Z 189,A 39.8942,B 1.7011,C 0.0251,E1 1.8281,E2 414.1002} C_DIS
LIN {X 107.7604,Y 89.7497,Z 189,A 40.982,B 1.7011,C 0.0241,E1 1.8263,E2 413.0577} C_DIS
LIN {X 105.1234,Y 92.8238,Z 189,A 42.6187,B 1.7011,C 0.0206,E1 1.8233,E2 411.4231} C_DIS
LIN {X 101.8883,Y 96.3638,Z 189,A 44.4103,B 1.7012,C 0.0174,E1 1.8199,E2 409.6522} C_DIS
LIN {X 98.7713,Y 99.5561,Z 189,A 46.2631,B 1.7012,C 0.0134,E1 1.8162,E2 407.7954} C_DIS
LIN {X 93.5551,Y 104.473,Z 189,A 48.6382,B 1.7012,C 0.0107,E1 1.8115,E2 405.4891} C_DIS
LIN {X 91.2449,Y 106.4973,Z 189,A 50.0797,B 1.7012,C 0.0071,E1 1.8084,E2 404.0245} C_DIS
LIN {X 87.8943,Y 109.2785,Z 189,A 51.7863,B 1.7013,C 0.0042,E1 1.8047,E2 402.3268} C_DIS
LIN {X 84.2281,Y 112.129,Z 189,A 53.5948,B 1.7013,C 0.0012,E1 1.8007,E2 400.5293} C_DIS
LIN {X 78.7826,Y 116.0195,Z 189,A 56.2776,B 1.7013,C -0.0034,E1 1.7946,E2 397.853} C_DIS
LIN {X 74.4869,Y 118.8237,Z 189,A 58.1534,B 1.7013,C -0.0057,E1 1.7902,E2 396.0044} C_DIS
LIN {X 70.7151,Y 121.1061,Z 189,A 59.9211,B 1.7013,C -0.0084,E1 1.786,E2 394.2409} C_DIS
LIN {X 66.6776,Y 123.375,Z 189,A 61.7353,B 1.7013,C -0.0109,E1 1.7816,E2 392.4365} C_DIS
LIN {X 62.4249,Y 125.5783,Z 189,A 63.6418,B 1.7013,C -0.0135,E1 1.7768,E2 390.5363} C_DIS
LIN {X 58.62,Y 127.3985,Z 189,A 65.1878,B 1.7013,C -0.015,E1 1.7729,E2 389.0123} C_DIS
LIN {X 55.3868,Y 128.8371,Z 189,A 66.5517,B 1.7013,C -0.0164,E1 1.7695,E2 387.6586} C_DIS
LIN {X 51.9028,Y 130.2806,Z 189,A 67.9895,B 1.7013,C -0.0179,E1 1.7658,E2 386.2336} C_DIS
LIN {X 48.8783,Y 131.4445,Z 189,A 69.2969,B 1.7012,C -0.0194,E1 1.7623,E2 384.9284} C_DIS
LIN {X 45.6524,Y 132.5994,Z 189,A 70.6494,B 1.7012,C -0.0208,E1 1.7588,E2 383.5819} C_DIS
LIN {X 42.6244,Y 133.6032,Z 189,A 73.0496,B 1.7011,C -0.0274,E1 1.752,E2 381.0475} C_DIS
LIN {X 34.7698,Y 135.8595,Z 189,A 74.9553,B 1.7011,C -0.0239,E1 1.7473,E2 379.3181} C_DIS
LIN {X 30.3163,Y 136.9225,Z 189,A 77.2193,B 1.7011,C -0.0273,E1 1.741,E2 377.007} C_DIS
LIN {X 27.1835,Y 137.5805,Z 189,A 78.2426,B 1.7011,C -0.027,E1 1.7383,E2 376.0187} C_DIS
LIN {X 24.2211,Y 138.1314,Z 189,A 79.5571,B 1.7011,C -0.0283,E1 1.7346,E2 374.6944} C_DIS
LIN {X 19.9364,Y 138.8138,Z 189,A 81.268,B 1.7011,C -0.0292,E1 1.7299,E2 372.9915} C_DIS
LIN {X 16.2754,Y 139.2909,Z 189,A 82.7019,B 1.7011,C -0.0298,E1 1.7259,E2 371.5671} C_DIS
LIN {X 12.0983,Y 139.7156,Z 189,A 84.4207,B 1.7011,C -0.0307,E1 1.7211,E2 369.8485} C_DIS
LIN {X 8.3275,Y 139.991,Z 189,A 85.8848,B 1.7011,C -0.031,E1 1.7171,E2 368.3947} C_DIS
LIN {X 4.514,Y 140.1669,Z 189,A 87.5055,B 1.7011,C -0.0318,E1 1.7125,E2 366.7673} C_DIS
LIN {X 0.7206,Y 140.2364,Z 189,A 88.9639,B 1.7011,C -0.0319,E1 1.7085,E2 365.3204} C_DIS
LIN {X -2.5313,Y 140.2156,Z 189,A 90.2491,B 1.7011,C -0.032,E1 1.7049,E2 364.0411} C_DIS
LIN {X -6.0296,Y 140.1097,Z 189,A 91.8561,B 1.701,C -0.0329,E1 1.7003,E2 362.4134} C_DIS
LIN {X -10.2495,Y 139.8631,Z 189,A 93.4499,B 1.701,C -0.0325,E1 1.6959,E2 360.8363} C_DIS
LIN {X -13.7534,Y 139.5625,Z 189,A 94.894,B 1.701,C -0.0325,E1 1.6919,E2 359.392} C_DIS
LIN {X -17.7248,Y 139.1144,Z 189,A 96.7288,B 1.701,C -0.0331,E1 1.6867,E2 357.5336} C_DIS
LIN {X -23.7257,Y 138.218,Z 189,A 98.9732,B 1.701,C -0.0318,E1 1.6806,E2 355.3187} C_DIS
LIN {X -26.523,Y 137.7072,Z 189,A 100.2252,B 1.701,C -0.0318,E1 1.6771,E2 354.0564} C_DIS
LIN {X -30.0976,Y 136.9711,Z 189,A 101.7719,B 1.701,C -0.0315,E1 1.6728,E2 352.5038} C_DIS
LIN {X -33.3397,Y 136.2181,Z 189,A 103.0603,B 1.701,C -0.0307,E1 1.6693,E2 351.2247} C_DIS
LIN {X -36.2163,Y 135.4808,Z 189,A 104.2934,B 1.701,C -0.0302,E1 1.666,E2 349.9898} C_DIS
LIN {X -39.8239,Y 134.4652,Z 189,A 105.8275,B 1.701,C -0.0294,E1 1.6618,E2 348.4562} C_DIS
LIN {X -42.9533,Y 133.4981,Z 189,A 107.2246,B 1.701,C -0.0287,E1 1.6581,E2 347.0527} C_DIS
LIN {X -46.4276,Y 132.3306,Z 189,A 108.7325,B 1.701,C -0.0277,E1 1.6541,E2 345.5444} C_DIS
LIN {X -49.4962,Y 131.2131,Z 189,A 110.1216,B 1.701,C -0.0269,E1 1.6504,E2 344.1494} C_DIS
LIN {X -52.7055,Y 129.9571,Z 189,A 112.0042,B 1.701,C -0.0269,E1 1.6454,E2 342.2102} C_DIS
LIN {X -56.5438,Y 128.3347,Z 189,A 113.4092,B 1.7011,C -0.0247,E1 1.6419,E2 340.8423} C_DIS
LIN {X -60.7557,Y 126.3941,Z 189,A 115.3581,B 1.7011,C -0.023,E1 1.6369,E2 338.888} C_DIS
LIN {X -64.0633,Y 124.7507,Z 189,A 116.8204,B 1.7011,C -0.0212,E1 1.6333,E2 337.4323} C_DIS
LIN {X -67.4714,Y 122.9428,Z 189,A 118.7889,B 1.7011,C -0.0204,E1 1.6283,E2 335.4172} C_DIS
LIN {X -70.5149,Y 121.2226,Z 189,A 120.0165,B 1.7012,C -0.0182,E1 1.6254,E2 334.2149} C_DIS
LIN {X -74.7532,Y 118.6556,Z 189,A 122.007,B 1.7012,C -0.0155,E1 1.6207,E2 332.2298} C_DIS
LIN {X -77.971,Y 116.5664,Z 189,A 123.9225,B 1.7012,C -0.0141,E1 1.6161,E2 330.273} C_DIS
LIN {X -82.3735,Y 113.498,Z 189,A 125.7947,B 1.7012,C -0.0103,E1 1.6119,E2 328.4412} C_DIS
LIN {X -84.8633,Y 111.6493,Z 189,A 127.4244,B 1.7012,C -0.0091,E1 1.6081,E2 326.7682} C_DIS
LIN {X -88.457,Y 108.824,Z 189,A 129.378,B 1.7012,C -0.0063,E1 1.6039,E2 324.8053} C_DIS
LIN {X -91.9551,Y 105.8846,Z 189,A 131.3226,B 1.7013,C -0.0033,E1 1.5997,E2 322.8524} C_DIS
LIN {X -95.2822,Y 102.9011,Z 189,A 133.2703,B 1.7013,C -0.0003,E1 1.5956,E2 320.891} C_DIS
LIN {X -98.5999,Y 99.7264,Z 189,A 135.2669,B 1.7013,C 0.0029,E1 1.5916,E2 318.8809} C_DIS
LIN {X -101.7623,Y 96.4974,Z 189,A 137.2125,B 1.7013,C 0.0063,E1 1.5878,E2 316.9242} C_DIS
LIN {X -104.8484,Y 93.1349,Z 189,A 139.1837,B 1.7013,C 0.0098,E1 1.5841,E2 314.9412} C_DIS
LIN {X -107.7857,Y 89.7192,Z 189,A 141.1118,B 1.7013,C 0.0134,E1 1.5806,E2 313.0036} C_DIS
LIN {X -110.5649,Y 86.2716,Z 189,A 143.1701,B 1.7013,C 0.0169,E1 1.577,E2 310.9156} C_DIS
LIN {X -114.8474,Y 80.4826,Z 189,A 146.7017,B 1.7012,C 0.0225,E1 1.5711,E2 307.3123} C_DIS
LIN {X -117.4778,Y 76.5912,Z 189,A 148.3013,B 1.7011,C 0.0273,E1 1.5687,E2 305.7541} C_DIS
LIN {X -121.7231,Y 69.6469,Z 189,A 151.4835,B 1.7009,C 0.0352,E1 1.5641,E2 302.5922} C_DIS
LIN {X -123.9354,Y 65.6266,Z 189,A 153.8294,B 1.7009,C 0.0392,E1 1.5609,E2 300.1886} C_DIS
LIN {X -125.6319,Y 62.3163,Z 189,A 155.8332,B 1.7008,C 0.0425,E1 1.5583,E2 298.1246} C_DIS
LIN {X -127.2832,Y 58.8694,Z 189,A 157.1185,B 1.7007,C 0.0466,E1 1.5569,E2 296.8754} C_DIS
LIN {X -129.9918,Y 52.6193,Z 189,A 160.0336,B 1.7005,C 0.0536,E1 1.5537,E2 293.9457} C_DIS
LIN {X -131.1936,Y 49.5481,Z 189,A 161.642,B 1.7004,C 0.0568,E1 1.552,E2 292.305} C_DIS
LIN {X -132.7282,Y 45.2809,Z 189,A 163.5713,B 1.7002,C 0.0616,E1 1.5502,E2 290.3673} C_DIS
LIN {X -133.675,Y 42.3996,Z 189,A 164.9295,B 1.7001,C 0.0648,E1 1.549,E2 288.9946} C_DIS
LIN {X -134.7709,Y 38.7799,Z 189,A 166.5885,B 1.6999,C 0.0688,E1 1.5477,E2 287.3221} C_DIS
LIN {X -136.2755,Y 33.1017,Z 189,A 169.3982,B 1.6997,C 0.075,E1 1.5457,E2 284.4614} C_DIS
LIN {X -137.3982,Y 28.079,Z 189,A 171.5856,B 1.6994,C 0.0807,E1 1.5444,E2 282.2644} C_DIS
LIN {X -138.1853,Y 23.9199,Z 189,A 174.0738,B 1.6992,C 0.0849,E1 1.5432,E2 279.6787} C_DIS
LIN {X -138.9559,Y 18.9342,Z 189,A 176.1974,B 1.6989,C 0.0905,E1 1.5424,E2 277.5481} C_DIS
LIN {X -139.4758,Y 14.6075,Z 189,A 177.5938,B 1.6986,C 0.0958,E1 1.542,E2 276.203} C_DIS
LIN {X -139.8324,Y 10.6699,Z 189,A -179.6636,B 1.6984,C 0.0994,E1 1.5414,E2 273.3131} C_DIS
LIN {X -140.1784,Y 4.1016,Z 189,A -177.9616,B 1.6979,C 0.1077,E1 1.5412,E2 271.7428} C_DIS
LIN {X -140.2015,Y -3.2693,Z 189,A -174.5007,B 1.6974,C 0.1158,E1 1.5412,E2 268.225} C_DIS
LIN {X -139.797,Y -11.1348,Z 189,A -170.7919,B 1.6968,C 0.1244,E1 1.5418,E2 264.4532} C_DIS
LIN {X -139.297,Y -16.2241,Z 189,A -168.8038,B 1.6963,C 0.1303,E1 1.5424,E2 262.4798} C_DIS
LIN {X -138.3105,Y -23.1716,Z 189,A -165.8673,B 1.6957,C 0.1382,E1 1.5436,E2 259.5356} C_DIS
LIN {X -137.4142,Y -28.0005,Z 189,A -163.2984,B 1.6953,C 0.1432,E1 1.5449,E2 256.8927} C_DIS
LIN {X -136.6888,Y -31.3506,Z 189,A -161.7679,B 1.695,C 0.1469,E1 1.5458,E2 255.3454} C_DIS
LIN {X -135.8245,Y -34.9079,Z 189,A -160.1641,B 1.6946,C 0.1508,E1 1.5469,E2 253.7278} C_DIS
LIN {X -135.0048,Y -37.9525,Z 189,A -158.7048,B 1.6943,C 0.1541,E1 1.548,E2 252.246} C_DIS
LIN {X -133.956,Y -41.5052,Z 189,A -156.9754,B 1.694,C 0.1579,E1 1.5495,E2 250.488} C_DIS
LIN {X -132.8526,Y -44.9125,Z 189,A -154.8979,B 1.6937,C 0.161,E1 1.5514,E2 248.3275} C_DIS
LIN {X -131.2359,Y -49.4352,Z 189,A -153.3743,B 1.6931,C 0.1666,E1 1.5528,E2 246.8646} C_DIS
LIN {X -129.8788,Y -52.8998,Z 189,A -151.5815,B 1.6928,C 0.1701,E1 1.5547,E2 245.0353} C_DIS
LIN {X -128.4546,Y -56.2715,Z 189,A -149.9996,B 1.6924,C 0.1738,E1 1.5565,E2 243.4421} C_DIS
LIN {X -126.4137,Y -60.7147,Z 189,A -147.9475,B 1.6919,C 0.1787,E1 1.5589,E2 241.3832} C_DIS
LIN {X -124.6757,Y -64.2106,Z 189,A -146.0864,B 1.6915,C 0.1822,E1 1.5613,E2 239.4861} C_DIS
LIN {X -122.4124,Y -68.4287,Z 189,A -144.0165,B 1.691,C 0.1867,E1 1.5641,E2 237.4012} C_DIS
LIN {X -120.1211,Y -72.3751,Z 189,A -141.8634,B 1.6906,C 0.1906,E1 1.5673,E2 235.2087} C_DIS
LIN {X -117.2833,Y -76.8888,Z 189,A -139.7165,B 1.69,C 0.1956,E1 1.5705,E2 233.0667} C_DIS
LIN {X -115.1782,Y -80.0073,Z 189,A -138.0485,B 1.6897,C 0.1987,E1 1.5732,E2 231.381} C_DIS
LIN {X -109.099,Y -88.1169,Z 189,A -133.9275,B 1.6886,C 0.2075,E1 1.5802,E2 227.2639} C_DIS
LIN {X -107.1862,Y -90.4347,Z 189,A -132.2239,B 1.6884,C 0.2091,E1 1.5833,E2 225.4942} C_DIS
LIN {X -103.4944,Y -94.6373,Z 189,A -129.9331,B 1.6879,C 0.2136,E1 1.5876,E2 223.2031} C_DIS
LIN {X -100.4907,Y -97.8209,Z 189,A -126.5642,B 1.6879,C 0.2136,E1 1.5947,E2 219.6108} C_DIS
LIN {X -93.4557,Y -104.562,Z 189,A -123.4734,B 1.6867,C 0.2224,E1 1.6008,E2 216.6471} C_DIS
LIN {X -90.457,Y -107.1675,Z 189,A -122.3553,B 1.6862,C 0.2262,E1 1.603,E2 215.6002} C_DIS
LIN {X -86.6034,Y -110.3042,Z 189,A -119.9864,B 1.6859,C 0.2286,E1 1.6083,E2 213.1836} C_DIS
LIN {X -82.1549,Y -113.6564,Z 189,A -117.6483,B 1.6854,C 0.2318,E1 1.6136,E2 210.8367} C_DIS
LIN {X -78.7515,Y -116.0405,Z 189,A -115.9884,B 1.6851,C 0.2342,E1 1.6174,E2 209.1821} C_DIS
LIN {X -75.8926,Y -117.9305,Z 189,A -114.3603,B 1.6849,C 0.2355,E1 1.6213,E2 207.5216} C_DIS
LIN {X -72.0877,Y -120.294,Z 189,A -112.4799,B 1.6846,C 0.2376,E1 1.6258,E2 205.6339} C_DIS
LIN {X -68.3044,Y -122.4821,Z 189,A -110.596,B 1.6844,C 0.2394,E1 1.6304,E2 203.7359} C_DIS
LIN {X -64.0388,Y -124.7632,Z 189,A -108.638,B 1.6841,C 0.2415,E1 1.6353,E2 201.7801} C_DIS
LIN {X -60.1475,Y -126.6847,Z 189,A -106.8221,B 1.6838,C 0.2432,E1 1.6399,E2 199.9578} C_DIS
LIN {X -57.0756,Y -128.0977,Z 189,A -105.3986,B 1.6837,C 0.2443,E1 1.6435,E2 198.528} C_DIS
LIN {X -53.7189,Y -129.5416,Z 189,A -103.8796,B 1.6835,C 0.2455,E1 1.6475,E2 197.0051} C_DIS
LIN {X -50.626,Y -130.781,Z 189,A -102.4856,B 1.6834,C 0.2464,E1 1.6511,E2 195.6061} C_DIS
LIN {X -47.0749,Y -132.1017,Z 189,A -100.8479,B 1.6833,C 0.2472,E1 1.6555,E2 193.9552} C_DIS
LIN {X -37.0523,Y -135.2566,Z 189,A -96.5714,B 1.6829,C 0.2497,E1 1.6669,E2 189.6802} C_DIS
LIN {X -30.1289,Y -136.9643,Z 189,A -93.6994,B 1.6827,C 0.2509,E1 1.6747,E2 186.8133} C_DIS
LIN {X -27.3682,Y -137.5429,Z 189,A -92.3072,B 1.6827,C 0.2503,E1 1.6786,E2 185.3863} C_DIS
LIN {X -22.9841,Y -138.3418,Z 189,A -90.5839,B 1.6827,C 0.2511,E1 1.6834,E2 183.6763} C_DIS
LIN {X -19.5198,Y -138.8733,Z 189,A -89.159,B 1.6827,C 0.2513,E1 1.6873,E2 182.2518} C_DIS
LIN {X -16.2927,Y -139.2888,Z 189,A -87.7462,B 1.6827,C 0.2511,E1 1.6913,E2 180.8265} C_DIS
LIN {X -11.8534,Y -139.7363,Z 189,A -85.9873,B 1.6827,C 0.2513,E1 1.6962,E2 179.076} C_DIS
LIN {X -7.8064,Y -140.0229,Z 189,A -84.2162,B 1.6827,C 0.2506,E1 1.7012,E2 177.2879} C_DIS
LIN {X -3.736,Y -140.1886,Z 189,A -82.6575,B 1.6827,C 0.2508,E1 1.7055,E2 175.7435} C_DIS
LIN {X 0.9853,Y -140.2333,Z 189,A -80.8791,B 1.6827,C 0.251,E1 1.7104,E2 173.9857} C_DIS
Enddeposition()
LIN {X 0.9853,Y -140.2333,Z 189,A -80.8791,B 1.6827,C 0.251,E1 1.7104,E2 173.9857} C_DIS
Startdeposition()
$VEL.CP = VEL_PRINT
LIN {X -0.0877,Y -141.1391,Z 189,A -81.8897,B 1.6738,C 0.2541,E1 1.6989,E2 175.1093} C_DIS
LIN {X -4.0805,Y -141.0785,Z 189,A -83.4731,B 1.6738,C 0.2543,E1 1.6945,E2 176.688} C_DIS
LIN {X -8.5273,Y -140.8796,Z 189,A -85.207,B 1.6738,C 0.2543,E1 1.6896,E2 178.4123} C_DIS
LIN {X -12.1347,Y -140.6149,Z 189,A -86.6529,B 1.6738,C 0.2542,E1 1.6856,E2 179.8557} C_DIS
LIN {X -16.3146,Y -140.1917,Z 189,A -88.4019,B 1.6738,C 0.2543,E1 1.6807,E2 181.6116} C_DIS
LIN {X -19.9376,Y -139.7219,Z 189,A -89.866,B 1.6738,C 0.2541,E1 1.6766,E2 183.0735} C_DIS
LIN {X -23.4302,Y -139.1789,Z 189,A -91.3043,B 1.6738,C 0.2539,E1 1.6727,E2 184.5129} C_DIS
LIN {X -27.0103,Y -138.5294,Z 189,A -92.7814,B 1.6738,C 0.2535,E1 1.6686,E2 185.9906} C_DIS
LIN {X -31.0148,Y -137.6879,Z 189,A -94.9286,B 1.6737,C 0.2548,E1 1.6625,E2 188.2075} C_DIS
LIN {X -35.3297,Y -136.6451,Z 189,A -96.2563,B 1.674,C 0.2523,E1 1.6591,E2 189.4685} C_DIS
LIN {X -38.9931,Y -135.6454,Z 189,A -98.4382,B 1.6738,C 0.2538,E1 1.653,E2 191.7418} C_DIS
LIN {X -43.8415,Y -134.1573,Z 189,A -100.1615,B 1.6742,C 0.2514,E1 1.6485,E2 193.4181} C_DIS
LIN {X -48.0596,Y -132.7025,Z 189,A -101.8011,B 1.6744,C 0.2496,E1 1.6442,E2 195.0337} C_DIS
LIN {X -51.4829,Y -131.4126,Z 189,A -103.3159,B 1.6746,C 0.2486,E1 1.6402,E2 196.5532} C_DIS
LIN {X -54.7035,Y -130.1048,Z 189,A -104.7729,B 1.6747,C 0.2476,E1 1.6364,E2 198.017} C_DIS
LIN {X -58.8033,Y -128.3044,Z 189,A -106.6697,B 1.6749,C 0.2462,E1 1.6315,E2 199.9253} C_DIS
LIN {X -62.7331,Y -126.4289,Z 189,A -108.4801,B 1.6752,C 0.2446,E1 1.627,E2 201.7421} C_DIS
LIN {X -67.4039,Y -124.0038,Z 189,A -110.7582,B 1.6755,C 0.2427,E1 1.6213,E2 204.0406} C_DIS
LIN {X -71.4867,Y -121.6956,Z 189,A -112.716,B 1.6757,C 0.2407,E1 1.6165,E2 206.0062} C_DIS
LIN {X -75.5204,Y -119.2346,Z 189,A -114.6742,B 1.6761,C 0.2384,E1 1.6118,E2 207.9703} C_DIS
LIN {X -79.3083,Y -116.7494,Z 189,A -116.6536,B 1.6764,C 0.2363,E1 1.6072,E2 209.9695} C_DIS
LIN {X -82.1785,Y -114.747,Z 189,A -118.3929,B 1.6765,C 0.235,E1 1.6031,E2 211.7537} C_DIS
LIN {X -85.227,Y -112.5016,Z 189,A -119.7013,B 1.6769,C 0.2322,E1 1.6002,E2 213.03} C_DIS
LIN {X -88.7774,Y -109.7215,Z 189,A -121.6393,B 1.6773,C 0.2296,E1 1.596,E2 214.9831} C_DIS
LIN {X -92.9326,Y -106.225,Z 189,A -123.9568,B 1.6778,C 0.2263,E1 1.591,E2 217.3164} C_DIS
LIN {X -96.4134,Y -103.0763,Z 189,A -126.7669,B 1.6779,C 0.2249,E1 1.585,E2 220.2524} C_DIS
LIN {X -101.0439,Y -98.5417,Z 189,A -128.4548,B 1.6788,C 0.2182,E1 1.5819,E2 221.8088} C_DIS
LIN {X -104.4679,Y -94.9033,Z 189,A -130.9058,B 1.6792,C 0.2151,E1 1.5771,E2 224.3186} C_DIS
LIN {X -108.1758,Y -90.6542,Z 189,A -133.301,B 1.6798,C 0.2108,E1 1.5727,E2 226.7282} C_DIS
LIN {X -114.4495,Y -82.5927,Z 189,A -137.47,B 1.6808,C 0.2022,E1 1.5656,E2 230.8997} C_DIS
LIN {X -117.4225,Y -78.308,Z 189,A -139.9656,B 1.6813,C 0.1981,E1 1.5616,E2 233.4471} C_DIS
LIN {X -119.824,Y -74.5814,Z 189,A -141.9363,B 1.6818,C 0.1942,E1 1.5586,E2 235.441} C_DIS
LIN {X -122.0708,Y -70.8444,Z 189,A -143.8642,B 1.6822,C 0.1904,E1 1.5558,E2 237.39} C_DIS
LIN {X -124.1836,Y -67.0725,Z 189,A -145.783,B 1.6826,C 0.1864,E1 1.5532,E2 239.3307} C_DIS
LIN {X -125.938,Y -63.7129,Z 189,A -147.3419,B 1.6831,C 0.1827,E1 1.5512,E2 240.8917} C_DIS
LIN {X -127.7112,Y -60.084,Z 189,A -149.0831,B 1.6835,C 0.1788,E1 1.5491,E2 242.6463} C_DIS
LIN {X -128.985,Y -57.2941,Z 189,A -150.7666,B 1.6837,C 0.1762,E1 1.5471,E2 244.3891} C_DIS
LIN {X -130.3244,Y -54.1777,Z 189,A -151.5058,B 1.6842,C 0.172,E1 1.5464,E2 245.0408} C_DIS
LIN {X -130.9984,Y -52.5272,Z 189,A -152.7214,B 1.6843,C 0.1707,E1 1.545,E2 246.3233} C_DIS
LIN {X -132.1523,Y -49.5521,Z 189,A -154.1056,B 1.6846,C 0.1675,E1 1.5436,E2 247.719} C_DIS
LIN {X -134.2895,Y -43.4307,Z 189,A -156.8344,B 1.6853,C 0.1608,E1 1.5411,E2 250.4599} C_DIS
LIN {X -135.1756,Y -40.5928,Z 189,A -158.4518,B 1.6856,C 0.1579,E1 1.5398,E2 252.1322} C_DIS
LIN {X -136.3489,Y -36.4506,Z 189,A -160.1758,B 1.686,C 0.1533,E1 1.5385,E2 253.8521} C_DIS
LIN {X -137.2339,Y -32.9627,Z 189,A -161.7754,B 1.6863,C 0.1494,E1 1.5374,E2 255.4697} C_DIS
LIN {X -138.0165,Y -29.5164,Z 189,A -163.3579,B 1.6867,C 0.1457,E1 1.5364,E2 257.0713} C_DIS
LIN {X -138.7427,Y -25.8949,Z 189,A -164.9222,B 1.687,C 0.1416,E1 1.5356,E2 258.6436} C_DIS
LIN {X -139.5716,Y -20.9696,Z 189,A -167.2465,B 1.6874,C 0.1363,E1 1.5345,E2 261.0064} C_DIS
LIN {X -140.167,Y -16.5224,Z 189,A -170.0867,B 1.6878,C 0.1321,E1 1.5336,E2 263.9798} C_DIS
LIN {X -140.7663,Y -10.2277,Z 189,A -172.4877,B 1.6883,C 0.1247,E1 1.533,E2 266.3577} C_DIS
LIN {X -141.0143,Y -5.9084,Z 189,A -173.7195,B 1.6887,C 0.1195,E1 1.5329,E2 267.5196} C_DIS
LIN {X -141.1305,Y -1.5925,Z 189,A -176.3643,B 1.689,C 0.1152,E1 1.5328,E2 270.2804} C_DIS
LIN {X -141.1099,Y 2.8308,Z 189,A -177.8399,B 1.6894,C 0.1099,E1 1.5328,E2 271.7133} C_DIS
LIN {X -140.8332,Y 9.2811,Z 189,A 179.2477,B 1.6898,C 0.1028,E1 1.5332,E2 274.6621} C_DIS
LIN {X -140.4774,Y 13.6324,Z 189,A 177.4138,B 1.6901,C 0.0979,E1 1.5337,E2 276.5029} C_DIS
LIN {X -140.0788,Y 17.2614,Z 189,A 175.8106,B 1.6903,C 0.0939,E1 1.5342,E2 278.1208} C_DIS
LIN {X -139.6143,Y 20.6877,Z 189,A 173.8318,B 1.6905,C 0.0904,E1 1.535,E2 280.1729} C_DIS
LIN {X -138.9946,Y 24.5017,Z 189,A 172.756,B 1.6908,C 0.0857,E1 1.5355,E2 281.1842} C_DIS
LIN {X -137.6105,Y 31.3534,Z 189,A 169.7767,B 1.6911,C 0.0781,E1 1.5372,E2 284.1801} C_DIS
LIN {X -136.5143,Y 35.8306,Z 189,A 167.3744,B 1.6913,C 0.0734,E1 1.5388,E2 286.6494} C_DIS
LIN {X -135.73,Y 38.6981,Z 189,A 166.0977,B 1.6915,C 0.0702,E1 1.5398,E2 287.9342} C_DIS
LIN {X -134.5371,Y 42.6556,Z 189,A 164.2716,B 1.6917,C 0.0659,E1 1.5413,E2 289.778} C_DIS
LIN {X -133.0886,Y 46.9861,Z 189,A 162.2717,B 1.6918,C 0.0611,E1 1.5431,E2 291.7953} C_DIS
LIN {X -132.0818,Y 49.7401,Z 189,A 160.9945,B 1.6919,C 0.0581,E1 1.5444,E2 293.0826} C_DIS
LIN {X -130.8856,Y 52.8071,Z 189,A 159.3315,B 1.692,C 0.0549,E1 1.5462,E2 294.7859} C_DIS
LIN {X -128.984,Y 57.2964,Z 189,A 157.168,B 1.6922,C 0.0501,E1 1.5486,E2 296.9712} C_DIS
LIN {X -126.5473,Y 62.4931,Z 189,A 155.2299,B 1.6924,C 0.0439,E1 1.5509,E2 298.8584} C_DIS
LIN {X -125.1298,Y 65.286,Z 189,A 153.4624,B 1.6924,C 0.0413,E1 1.5532,E2 300.6874} C_DIS
LIN {X -123.0326,Y 69.1604,Z 189,A 150.887,B 1.6925,C 0.0378,E1 1.5568,E2 303.3594} C_DIS
LIN {X -120.4064,Y 73.6376,Z 189,A 149.5589,B 1.6926,C 0.0321,E1 1.5586,E2 304.5893} C_DIS
LIN {X -117.6674,Y 77.9404,Z 189,A 146.7311,B 1.6927,C 0.0282,E1 1.563,E2 307.5097} C_DIS
LIN {X -115.7339,Y 80.783,Z 189,A 145.5663,B 1.6927,C 0.0248,E1 1.5648,E2 308.6451} C_DIS
LIN {X -111.8512,Y 86.0794,Z 189,A 142.6214,B 1.6928,C 0.0195,E1 1.5698,E2 311.6226} C_DIS
LIN {X -109.1424,Y 89.4883,Z 189,A 140.7487,B 1.6928,C 0.0159,E1 1.5731,E2 313.507} C_DIS
LIN {X -106.2227,Y 92.9351,Z 189,A 138.787,B 1.6928,C 0.0124,E1 1.5767,E2 315.4831} C_DIS
LIN {X -103.1247,Y 96.3615,Z 189,A 136.8001,B 1.6929,C 0.0089,E1 1.5805,E2 317.4824} C_DIS
LIN {X -100.1733,Y 99.4258,Z 189,A 134.9527,B 1.6929,C 0.0058,E1 1.5841,E2 319.3433} C_DIS
LIN {X -96.8429,Y 102.6724,Z 189,A 132.9859,B 1.6929,C 0.0026,E1 1.5881,E2 321.3184} C_DIS
LIN {X -93.5763,Y 105.6583,Z 189,A 131.0582,B 1.6929,C -0.0003,E1 1.5922,E2 323.2608} C_DIS
LIN {X -90.0817,Y 108.653,Z 189,A 129.0915,B 1.6929,C -0.0032,E1 1.5964,E2 325.2382} C_DIS
LIN {X -86.4253,Y 111.5833,Z 189,A 127.0968,B 1.6929,C -0.0061,E1 1.6008,E2 327.2429} C_DIS
LIN {X -82.6834,Y 114.3839,Z 189,A 124.8424,B 1.6929,C -0.0082,E1 1.606,E2 329.539} C_DIS
LIN {X -79.6925,Y 116.4874,Z 189,A 123.5861,B 1.6929,C -0.0108,E1 1.6088,E2 330.7669} C_DIS
LIN {X -75.8812,Y 119.0054,Z 189,A 121.6221,B 1.6929,C -0.013,E1 1.6135,E2 332.743} C_DIS
LIN {X -72.08,Y 121.3453,Z 189,A 119.1736,B 1.6929,C -0.0139,E1 1.6196,E2 335.2665} C_DIS
LIN {X -67.5185,Y 123.9413,Z 189,A 117.8213,B 1.6929,C -0.0181,E1 1.6226,E2 336.5243} C_DIS
LIN {X -64.7788,Y 125.3954,Z 189,A 116.0448,B 1.6929,C -0.0183,E1 1.6272,E2 338.3621} C_DIS
LIN {X -59.7826,Y 127.8515,Z 189,A 114.0945,B 1.6929,C -0.0213,E1 1.632,E2 340.274} C_DIS
LIN {X -57.2336,Y 129.0121,Z 189,A 112.3912,B 1.6929,C -0.0209,E1 1.6366,E2 342.0443} C_DIS
LIN {X -53.4273,Y 130.6356,Z 189,A 111.1577,B 1.6928,C -0.0235,E1 1.6396,E2 343.2235} C_DIS
LIN {X -50.723,Y 131.708,Z 189,A 109.8847,B 1.6928,C -0.0242,E1 1.643,E2 344.5069} C_DIS
LIN {X -47.2628,Y 132.9898,Z 189,A 108.3678,B 1.6928,C -0.0253,E1 1.647,E2 346.0252} C_DIS
LIN {X -44.4098,Y 133.9681,Z 189,A 107.1039,B 1.6928,C -0.026,E1 1.6503,E2 347.2931} C_DIS
LIN {X -40.9525,Y 135.0655,Z 189,A 105.5904,B 1.6928,C -0.0267,E1 1.6544,E2 348.8108} C_DIS
LIN {X -37.7109,Y 136.006,Z 189,A 104.1979,B 1.6928,C -0.0274,E1 1.6582,E2 350.2052} C_DIS
LIN {X -33.7561,Y 137.0427,Z 189,A 102.5945,B 1.6928,C -0.0283,E1 1.6625,E2 351.8011} C_DIS
LIN {X -30.8693,Y 137.7211,Z 189,A 101.3124,B 1.6927,C -0.0285,E1 1.666,E2 353.0919} C_DIS
LIN {X -27.4072,Y 138.4525,Z 189,A 99.8976,B 1.6927,C -0.029,E1 1.6699,E2 354.5034} C_DIS
LIN {X -23.0919,Y 139.2354,Z 189,A 98.0355,B 1.6927,C -0.0292,E1 1.6751,E2 356.3744} C_DIS
LIN {X -18.426,Y 139.9293,Z 189,A 95.7799,B 1.6927,C -0.0283,E1 1.6814,E2 358.6695} C_DIS
LIN {X -14.6334,Y 140.3774,Z 189,A 94.6581,B 1.6927,C -0.0299,E1 1.6844,E2 359.7396} C_DIS
LIN {X -11.521,Y 140.6668,Z 189,A 93.3625,B 1.6927,C -0.0298,E1 1.6881,E2 361.0378} C_DIS
LIN {X -7.8491,Y 140.921,Z 189,A 91.7339,B 1.6927,C -0.0292,E1 1.6927,E2 362.6819} C_DIS
LIN {X -3.9538,Y 141.082,Z 189,A 90.2897,B 1.6927,C -0.0294,E1 1.6967,E2 364.1088} C_DIS
LIN {X -0.6147,Y 141.1362,Z 189,A 88.9215,B 1.6927,C -0.0291,E1 1.7005,E2 365.478} C_DIS
LIN {X 3.3335,Y 141.0993,Z 189,A 87.2495,B 1.6927,C -0.0283,E1 1.7052,E2 367.1576} C_DIS
LIN {X 7.181,Y 140.9546,Z 189,A 85.742,B 1.6927,C -0.028,E1 1.7094,E2 368.6578} C_DIS
LIN {X 10.95,Y 140.7135,Z 189,A 84.1406,B 1.6927,C -0.027,E1 1.7139,E2 370.267} C_DIS
LIN {X 15.0782,Y 140.3295,Z 189,A 82.5713,B 1.6927,C -0.0266,E1 1.7183,E2 371.822} C_DIS
LIN {X 18.3652,Y 139.9373,Z 189,A 81.3058,B 1.6927,C -0.0261,E1 1.7217,E2 373.0777} C_DIS
LIN {X 21.8228,Y 139.44,Z 189,A 79.8888,B 1.6927,C -0.0252,E1 1.7257,E2 374.4941} C_DIS
LIN {X 25.7562,Y 138.7692,Z 189,A 78.3517,B 1.6927,C -0.0244,E1 1.7299,E2 376.0209} C_DIS
LIN {X 32.7291,Y 137.2902,Z 189,A 75.6712,B 1.6927,C -0.0229,E1 1.7372,E2 378.6749} C_DIS
LIN {X 41.2635,Y 134.9703,Z 189,A 71.9313,B 1.6928,C -0.0187,E1 1.7473,E2 382.4321} C_DIS
LIN {X 44.4058,Y 133.9694,Z 189,A 70.6529,B 1.6928,C -0.0176,E1 1.7507,E2 383.7028} C_DIS
LIN {X 48.2224,Y 132.6438,Z 189,A 69.1257,B 1.6928,C -0.0162,E1 1.7547,E2 385.2162} C_DIS
LIN {X 51.4694,Y 131.4179,Z 189,A 67.7327,B 1.6928,C -0.0146,E1 1.7583,E2 386.607} C_DIS
LIN {X 54.8088,Y 130.0609,Z 189,A 66.359,B 1.6928,C -0.0132,E1 1.7619,E2 387.9696} C_DIS
LIN {X 58.1019,Y 128.6237,Z 189,A 64.9685,B 1.6928,C -0.0116,E1 1.7654,E2 389.3516} C_DIS
LIN {X 60.9369,Y 127.304,Z 189,A 63.7524,B 1.6929,C -0.0101,E1 1.7685,E2 390.561} C_DIS
LIN {X 64.7788,Y 125.3954,Z 189,A 61.9335,B 1.6929,C -0.0071,E1 1.773,E2 392.3892} C_DIS
LIN {X 68.9299,Y 123.1622,Z 189,A 60.1231,B 1.6929,C -0.0047,E1 1.7775,E2 394.1869} C_DIS
LIN {X 73.0042,Y 120.7914,Z 189,A 58.3277,B 1.6929,C -0.0023,E1 1.7818,E2 395.9677} C_DIS
LIN {X 76.9643,Y 118.3076,Z 189,A 56.5146,B 1.6929,C 0.0004,E1 1.786,E2 397.7705} C_DIS
LIN {X 80.2482,Y 116.106,Z 189,A 54.8033,B 1.6929,C 0.0038,E1 1.79,E2 399.4947} C_DIS
LIN {X 82.917,Y 114.2145,Z 189,A 53.9589,B 1.6929,C 0.0035,E1 1.7918,E2 400.2798} C_DIS
LIN {X 85.4985,Y 112.2955,Z 189,A 52.4772,B 1.6929,C 0.0069,E1 1.7951,E2 401.7832} C_DIS
LIN {X 89.0529,Y 109.4983,Z 189,A 50.7251,B 1.6929,C 0.0099,E1 1.7989,E2 403.525} C_DIS
LIN {X 92.5875,Y 106.526,Z 189,A 49.0015,B 1.6929,C 0.0127,E1 1.8026,E2 405.2301} C_DIS
LIN {X 95.8733,Y 103.5793,Z 189,A 46.9188,B 1.6929,C 0.018,E1 1.8069,E2 407.3487} C_DIS
LIN {X 99.0832,Y 100.5128,Z 189,A 45.6566,B 1.6929,C 0.0185,E1 1.8093,E2 408.5445} C_DIS
LIN {X 102.0681,Y 97.4796,Z 189,A 43.9731,B 1.6928,C 0.0219,E1 1.8126,E2 410.2227} C_DIS
LIN {X 105.2653,Y 94.0182,Z 189,A 42.1661,B 1.6928,C 0.0255,E1 1.816,E2 412.0167} C_DIS
LIN {X 108.2807,Y 90.5291,Z 189,A 40.4022,B 1.6927,C 0.029,E1 1.8192,E2 413.7675} C_DIS
LIN {X 112.1306,Y 85.714,Z 189,A 38.2406,B 1.6927,C 0.0326,E1 1.8228,E2 415.8868} C_DIS
LIN {X 114.3759,Y 82.6943,Z 189,A 36.6074,B 1.6925,C 0.0368,E1 1.8256,E2 417.5336} C_DIS
LIN {X 116.8435,Y 79.1693,Z 189,A 34.7173,B 1.6925,C 0.0419,E1 1.8286,E2 419.4421} C_DIS
LIN {X 119.0876,Y 75.7527,Z 189,A 33.6606,B 1.6925,C 0.0421,E1 1.8301,E2 420.4233} C_DIS
LIN {X 120.7277,Y 73.1096,Z 189,A 32.291,B 1.6923,C 0.0458,E1 1.8321,E2 421.8068} C_DIS
LIN {X 123.0038,Y 69.2117,Z 189,A 30.5867,B 1.6923,C 0.0496,E1 1.8344,E2 423.4955} C_DIS
LIN {X 125.1982,Y 65.1559,Z 189,A 28.9112,B 1.6921,C 0.053,E1 1.8366,E2 425.1465} C_DIS
LIN {X 126.7891,Y 62.0029,Z 189,A 27.4813,B 1.692,C 0.0566,E1 1.8384,E2 426.5764} C_DIS
LIN {X 129.2764,Y 56.6365,Z 189,A 25.4311,B 1.6919,C 0.0605,E1 1.8407,E2 428.5826} C_DIS
LIN {X 130.323,Y 54.181,Z 189,A 24.3361,B 1.6917,C 0.0634,E1 1.8419,E2 429.6794} C_DIS
LIN {X 131.6507,Y 50.8705,Z 189,A 23.0238,B 1.6917,C 0.0663,E1 1.8432,E2 430.9749} C_DIS
LIN {X 132.8759,Y 47.5786,Z 189,A 21.7222,B 1.6915,C 0.0693,E1 1.8444,E2 432.261} C_DIS
LIN {X 134.0148,Y 44.2697,Z 189,A 20.3777,B 1.6914,C 0.0726,E1 1.8456,E2 433.5963} C_DIS
LIN {X 135.2555,Y 40.3246,Z 189,A 18.1045,B 1.691,C 0.0812,E1 1.8475,E2 435.9466} C_DIS
LIN {X 136.8634,Y 34.4695,Z 189,A 15.6797,B 1.6907,C 0.0876,E1 1.8492,E2 438.3673} C_DIS
LIN {X 138.4158,Y 27.5875,Z 189,A 13.9072,B 1.6907,C 0.088,E1 1.8501,E2 440.0004} C_DIS
LIN {X 139.2809,Y 22.8191,Z 189,A 12.1703,B 1.6904,C 0.0918,E1 1.8509,E2 441.7081} C_DIS
LIN {X 139.7399,Y 19.8119,Z 189,A 10.9599,B 1.6903,C 0.0951,E1 1.8514,E2 442.916} C_DIS
LIN {X 140.2379,Y 15.9275,Z 189,A 9.3243,B 1.69,C 0.0999,E1 1.852,E2 444.5585} C_DIS
LIN {X 140.6348,Y 11.8989,Z 189,A 7.9671,B 1.6898,C 0.1024,E1 1.8523,E2 445.879} C_DIS
LIN {X 140.8985,Y 8.2205,Z 189,A 6.6057,B 1.6896,C 0.1057,E1 1.8525,E2 447.2233} C_DIS
LIN {X 141.0416,Y 5.2067,Z 189,A 5.4304,B 1.6894,C 0.1088,E1 1.8527,E2 448.3928} C_DIS
LIN {X 141.1372,Y 0.6508,Z 189,A 3.7348,B 1.6892,C 0.1129,E1 1.8527,E2 450.0691} C_DIS
LIN {X 141.1051,Y -3.1169,Z 189,A 2.1969,B 1.6889,C 0.1172,E1 1.8527,E2 451.609} C_DIS
LIN {X 140.9466,Y -7.3411,Z 189,A 0.7233,B 1.6887,C 0.1203,E1 1.8525,E2 453.0514} C_DIS
LIN {X 140.6506,Y -11.7124,Z 189,A -0.9228,B 1.6884,C 0.1243,E1 1.8522,E2 454.681} C_DIS
LIN {X 140.3278,Y -15.0941,Z 189,A -2.2198,B 1.6881,C 0.1276,E1 1.8518,E2 455.9679} C_DIS
LIN {X 139.7885,Y -19.4717,Z 189,A -3.925,B 1.6878,C 0.132,E1 1.8512,E2 457.6628} C_DIS
LIN {X 139.1827,Y -23.4075,Z 189,A -5.3363,B 1.6875,C 0.135,E1 1.8506,E2 459.0477} C_DIS
LIN {X 138.4777,Y -27.2807,Z 189,A -6.7843,B 1.6873,C 0.1384,E1 1.8498,E2 460.4766} C_DIS
LIN {X 137.8416,Y -30.3262,Z 189,A -7.9313,B 1.6871,C 0.141,E1 1.8492,E2 461.6089} C_DIS
LIN {X 136.9786,Y -34.0156,Z 189,A -9.6839,B 1.6866,C 0.1468,E1 1.848,E2 463.3914} C_DIS
LIN {X 136.099,Y -37.3785,Z 189,A -10.6309,B 1.6866,C 0.1473,E1 1.8474,E2 464.2767} C_DIS
LIN {X 135.1758,Y -40.5919,Z 189,A -12.3197,B 1.686,C 0.1533,E1 1.846,E2 466.0113} C_DIS
LIN {X 134.0199,Y -44.2541,Z 189,A -13.5186,B 1.6858,C 0.155,E1 1.845,E2 467.1626} C_DIS
LIN {X 132.674,Y -48.1386,Z 189,A -14.9533,B 1.6856,C 0.1578,E1 1.8437,E2 468.5667} C_DIS
LIN {X 131.3768,Y -51.5751,Z 189,A -16.3325,B 1.6853,C 0.161,E1 1.8423,E2 469.9318} C_DIS
LIN {X 129.8551,Y -55.2979,Z 189,A -17.8775,B 1.6849,C 0.1647,E1 1.8406,E2 471.4661} C_DIS
LIN {X 128.3998,Y -58.597,Z 189,A -19.7318,B 1.6843,C 0.1712,E1 1.8384,E2 473.3746} C_DIS
LIN {X 126.2669,Y -63.0615,Z 189,A -21.0735,B 1.6843,C 0.1717,E1 1.8369,E2 474.6269} C_DIS
LIN {X 124.1644,Y -67.1077,Z 189,A -22.9562,B 1.6837,C 0.1766,E1 1.8344,E2 476.5153} C_DIS
LIN {X 122.4755,Y -70.1426,Z 189,A -24.7799,B 1.683,C 0.183,E1 1.8318,E2 478.3966} C_DIS
LIN {X 119.4712,Y -75.1456,Z 189,A -26.3248,B 1.683,C 0.1832,E1 1.8297,E2 479.8305} C_DIS
LIN {X 117.1882,Y -78.6589,Z 189,A -27.9838,B 1.6826,C 0.187,E1 1.8271,E2 481.4849} C_DIS
LIN {X 114.7296,Y -82.2029,Z 189,A -29.6221,B 1.6822,C 0.1904,E1 1.8245,E2 483.109} C_DIS
LIN {X 111.9615,Y -85.9352,Z 189,A -31.3968,B 1.6818,C 0.194,E1 1.8216,E2 484.8697} C_DIS
LIN {X 109.0436,Y -89.6092,Z 189,A -33.154,B 1.6814,C 0.1974,E1 1.8185,E2 486.608} C_DIS
LIN {X 106.1932,Y -92.9689,Z 189,A -34.8396,B 1.681,C 0.2007,E1 1.8155,E2 488.2806} C_DIS
LIN {X 103.1322,Y -96.3534,Z 189,A -36.5876,B 1.6806,C 0.204,E1 1.8122,E2 490.0154} C_DIS
LIN {X 100.0607,Y -99.5392,Z 189,A -38.2548,B 1.6802,C 0.207,E1 1.8089,E2 491.6659} C_DIS
LIN {X 96.9018,Y -102.6168,Z 189,A -39.9698,B 1.6798,C 0.2102,E1 1.8055,E2 493.3719} C_DIS
LIN {X 93.4798,Y -105.7435,Z 189,A -41.7236,B 1.6795,C 0.2132,E1 1.8019,E2 495.1091} C_DIS
LIN {X 90.0837,Y -108.6513,Z 189,A -43.457,B 1.6791,C 0.2162,E1 1.7982,E2 496.8325} C_DIS
LIN {X 86.4227,Y -111.5854,Z 189,A -45.2377,B 1.6787,C 0.2191,E1 1.7943,E2 498.5972} C_DIS
LIN {X 82.8819,Y -114.24,Z 189,A -46.9643,B 1.6783,C 0.2219,E1 1.7905,E2 500.3154} C_DIS
LIN {X 79.0598,Y -116.9176,Z 189,A -48.7426,B 1.678,C 0.2245,E1 1.7864,E2 502.0787} C_DIS
LIN {X 75.2007,Y -119.4364,Z 189,A -50.5377,B 1.6776,C 0.2273,E1 1.7822,E2 503.8645} C_DIS
LIN {X 71.1828,Y -121.8742,Z 189,A -52.3813,B 1.6773,C 0.23,E1 1.7778,E2 505.7005} C_DIS
LIN {X 64.5417,Y -125.5161,Z 189,A -55.1185,B 1.6769,C 0.2327,E1 1.7711,E2 508.3921} C_DIS
LIN {X 62.1031,Y -126.7397,Z 189,A -56.9125,B 1.6761,C 0.2382,E1 1.7664,E2 510.2839} C_DIS
LIN {X 57.1256,Y -129.0603,Z 189,A -58.4378,B 1.6762,C 0.2373,E1 1.7627,E2 511.7113} C_DIS
LIN {X 54.0705,Y -130.3692,Z 189,A -59.6982,B 1.6761,C 0.2386,E1 1.7595,E2 512.96} C_DIS
LIN {X 51.2373,Y -131.5081,Z 189,A -60.9657,B 1.6758,C 0.2403,E1 1.7562,E2 514.2324} C_DIS
LIN {X 47.2705,Y -132.987,Z 189,A -62.5533,B 1.6756,C 0.2416,E1 1.752,E2 515.8025} C_DIS
LIN {X 44.0745,Y -134.0798,Z 189,A -64.2793,B 1.6751,C 0.245,E1 1.7473,E2 517.5798} C_DIS
LIN {X 40.2822,Y -135.268,Z 189,A -65.4732,B 1.6751,C 0.2445,E1 1.7443,E2 518.7153} C_DIS
LIN {X 37.4339,Y -136.0835,Z 189,A -66.8499,B 1.6749,C 0.2466,E1 1.7405,E2 520.1174} C_DIS
LIN {X 31.7231,Y -137.5261,Z 189,A -68.7648,B 1.6749,C 0.2463,E1 1.7355,E2 521.966} C_DIS
LIN {X 25.357,Y -138.8415,Z 189,A -71.4098,B 1.6746,C 0.2485,E1 1.7282,E2 524.6136} C_DIS
LIN {X 22.139,Y -139.3911,Z 189,A -72.8993,B 1.6743,C 0.2503,E1 1.724,E2 526.1273} C_DIS
LIN {X 18.3282,Y -139.9421,Z 189,A -74.3922,B 1.6743,C 0.251,E1 1.7199,E2 527.6111} C_DIS
LIN {X 14.8213,Y -140.3572,Z 189,A -75.7594,B 1.6742,C 0.2515,E1 1.7161,E2 528.9696} C_DIS
LIN {X 11.7027,Y -140.6514,Z 189,A -77.0728,B 1.674,C 0.2523,E1 1.7124,E2 530.2897} C_DIS
LIN {X 7.3152,Y -140.9479,Z 189,A -78.8177,B 1.674,C 0.2529,E1 1.7075,E2 532.0298} C_DIS
LIN {X 3.9314,Y -141.0826,Z 189,A -80.1927,B 1.6739,C 0.2534,E1 1.7037,E2 533.4055} C_DIS
LIN {X 0.9912,Y -141.132,Z 189,A -81.0502,B 1.674,C 0.2523,E1 1.7014,E2 534.2155} C_DIS
Enddeposition()
LIN {X 0.9912,Y -141.132,Z 189,A -81.0502,B 1.674,C 0.2523,E1 1.7014,E2 534.2155} C_DIS
Startdeposition()
$VEL.CP = VEL_PRINT
LIN {X 3.0137,Y -142.0061,Z 189,A -79.9252,B 1.6743,C 0.2514,E1 1.7047,E2 533.0734} C_DIS
LIN {X 6.9809,Y -141.865,Z 189,A -78.2543,B 1.6745,C 0.2505,E1 1.7095,E2 531.3915} C_DIS
LIN {X 11.5524,Y -141.5665,Z 189,A -76.4686,B 1.6745,C 0.2499,E1 1.7144,E2 529.6139} C_DIS
LIN {X 15.5648,Y -141.1815,Z 189,A -74.7784,B 1.6747,C 0.2487,E1 1.7192,E2 527.9135} C_DIS
LIN {X 20.2963,Y -140.5789,Z 189,A -72.9539,B 1.6748,C 0.248,E1 1.7242,E2 526.1023} C_DIS
LIN {X 24.5704,Y -139.8958,Z 189,A -71.4343,B 1.6748,C 0.2479,E1 1.7283,E2 524.6145} C_DIS
LIN {X 28.5368,Y -139.1402,Z 189,A -69.3546,B 1.6754,C 0.2442,E1 1.7342,E2 522.4683} C_DIS
LIN {X 32.3367,Y -138.3082,Z 189,A -68.0494,B 1.6754,C 0.2442,E1 1.7377,E2 521.2006} C_DIS
LIN {X 36.7657,Y -137.1955,Z 189,A -66.3926,B 1.6754,C 0.2435,E1 1.7421,E2 519.5695} C_DIS
LIN {X 40.8889,Y -136.0253,Z 189,A -64.3057,B 1.676,C 0.2397,E1 1.7479,E2 517.4295} C_DIS
LIN {X 44.6655,Y -134.8306,Z 189,A -63.1157,B 1.676,C 0.2402,E1 1.7509,E2 516.2977} C_DIS
LIN {X 48.1898,Y -133.6114,Z 189,A -61.7503,B 1.6761,C 0.2392,E1 1.7544,E2 514.9513} C_DIS
LIN {X 51.32,Y -132.4407,Z 189,A -60.3942,B 1.6763,C 0.2375,E1 1.758,E2 513.5932} C_DIS
LIN {X 54.8573,Y -131.015,Z 189,A -58.6098,B 1.6768,C 0.2341,E1 1.7627,E2 511.772} C_DIS
LIN {X 58.138,Y -129.5925,Z 189,A -57.64,B 1.6768,C 0.2349,E1 1.765,E2 510.8697} C_DIS
LIN {X 60.895,Y -128.3205,Z 189,A -56.3968,B 1.677,C 0.2331,E1 1.7682,E2 509.6229} C_DIS
LIN {X 64.0882,Y -126.756,Z 189,A -54.9409,B 1.6773,C 0.2309,E1 1.7718,E2 508.1629} C_DIS
LIN {X 68.9594,Y -124.175,Z 189,A -52.78,B 1.6777,C 0.2278,E1 1.7772,E2 506.0095} C_DIS
LIN {X 72.9633,Y -121.8657,Z 189,A -50.9888,B 1.678,C 0.2253,E1 1.7815,E2 504.2275} C_DIS
LIN {X 76.7716,Y -119.503,Z 189,A -49.2745,B 1.6784,C 0.2228,E1 1.7855,E2 502.5253} C_DIS
LIN {X 80.5881,Y -116.9633,Z 189,A -47.5036,B 1.6787,C 0.2201,E1 1.7896,E2 500.7643} C_DIS
LIN {X 84.3347,Y -114.2915,Z 189,A -45.7329,B 1.6791,C 0.2172,E1 1.7936,E2 499.0045} C_DIS
LIN {X 88.0569,Y -111.4493,Z 189,A -43.9289,B 1.6795,C 0.2142,E1 1.7975,E2 497.2112} C_DIS
LIN {X 91.6475,Y -108.5161,Z 189,A -42.1604,B 1.6799,C 0.2113,E1 1.8013,E2 495.4559} C_DIS
LIN {X 95.1251,Y -105.4808,Z 189,A -40.3969,B 1.6802,C 0.2082,E1 1.805,E2 493.705} C_DIS
LIN {X 98.5067,Y -102.3298,Z 189,A -38.6444,B 1.6806,C 0.205,E1 1.8085,E2 491.9671} C_DIS
LIN {X 101.5925,Y -99.2665,Z 189,A -37.0096,B 1.681,C 0.2021,E1 1.8117,E2 490.3479} C_DIS
LIN {X 104.8221,Y -95.8502,Z 189,A -35.2175,B 1.6814,C 0.1987,E1 1.8151,E2 488.5692} C_DIS
LIN {X 107.9174,Y -92.3517,Z 189,A -33.4382,B 1.6818,C 0.1952,E1 1.8183,E2 486.8034} C_DIS
LIN {X 110.8893,Y -88.761,Z 189,A -31.686,B 1.6822,C 0.1918,E1 1.8214,E2 485.0678} C_DIS
LIN {X 113.7143,Y -85.1116,Z 189,A -29.9562,B 1.6826,C 0.1884,E1 1.8243,E2 483.3553} C_DIS
LIN {X 116.2729,Y -81.5815,Z 189,A -28.3237,B 1.6829,C 0.1851,E1 1.8269,E2 481.7392} C_DIS
LIN {X 118.8263,Y -77.8154,Z 189,A -26.6146,B 1.6833,C 0.1815,E1 1.8295,E2 480.0465} C_DIS
LIN {X 121.84,Y -73.006,Z 189,A -24.1858,B 1.684,C 0.1749,E1 1.8331,E2 477.5963} C_DIS
LIN {X 123.8555,Y -69.5315,Z 189,A -22.9934,B 1.6841,C 0.1739,E1 1.8346,E2 476.4629} C_DIS
LIN {X 126.124,Y -65.3268,Z 189,A -21.1296,B 1.6846,C 0.1694,E1 1.8371,E2 474.6065} C_DIS
LIN {X 127.4907,Y -62.6131,Z 189,A -19.8303,B 1.685,C 0.1658,E1 1.8387,E2 473.2959} C_DIS
LIN {X 128.9935,Y -59.4554,Z 189,A -18.866,B 1.685,C 0.1653,E1 1.8397,E2 472.3929} C_DIS
LIN {X 130.9547,Y -55.0017,Z 189,A -17.0387,B 1.6854,C 0.1611,E1 1.8418,E2 470.5831} C_DIS
LIN {X 132.3018,Y -51.6773,Z 189,A -15.5411,B 1.6858,C 0.1569,E1 1.8433,E2 469.0774} C_DIS
LIN {X 134.0218,Y -47.0394,Z 189,A -13.8986,B 1.6861,C 0.1541,E1 1.8448,E2 467.4823} C_DIS
LIN {X 136.2448,Y -40.1458,Z 189,A -11.075,B 1.6867,C 0.1469,E1 1.8472,E2 464.6704} C_DIS
LIN {X 137.065,Y -37.2546,Z 189,A -9.7452,B 1.6871,C 0.1428,E1 1.8482,E2 463.3237} C_DIS
LIN {X 138.3251,Y -32.2628,Z 189,A -7.9297,B 1.6874,C 0.139,E1 1.8494,E2 461.5427} C_DIS
LIN {X 139.1599,Y -28.44,Z 189,A -6.5998,B 1.6876,C 0.1364,E1 1.8501,E2 460.2458} C_DIS
LIN {X 139.7108,Y -25.604,Z 189,A -5.5956,B 1.6877,C 0.1343,E1 1.8506,E2 459.2629} C_DIS
LIN {X 140.3272,Y -21.9694,Z 189,A -4.0582,B 1.6881,C 0.1298,E1 1.8513,E2 457.7176} C_DIS
LIN {X 140.905,Y -17.901,Z 189,A -2.6078,B 1.6883,C 0.1267,E1 1.8518,E2 456.2945} C_DIS
LIN {X 141.2835,Y -14.6168,Z 189,A -1.2754,B 1.6886,C 0.123,E1 1.8522,E2 454.9614} C_DIS
LIN {X 141.6567,Y -10.3807,Z 189,A 0.2231,B 1.6888,C 0.1197,E1 1.8526,E2 453.4912} C_DIS
LIN {X 141.8988,Y -6.2997,Z 189,A 1.8478,B 1.6892,C 0.1153,E1 1.8528,E2 451.8689} C_DIS
LIN {X 142.0205,Y -2.147,Z 189,A 3.2502,B 1.6893,C 0.1126,E1 1.8528,E2 450.5024} C_DIS
LIN {X 142.0232,Y 1.9839,Z 189,A 4.8888,B 1.6896,C 0.1081,E1 1.8528,E2 448.8667} C_DIS
LIN {X 141.9075,Y 6.0772,Z 189,A 6.4656,B 1.6899,C 0.104,E1 1.8528,E2 447.299} C_DIS
LIN {X 141.6596,Y 10.3405,Z 189,A 7.9459,B 1.6901,C 0.1009,E1 1.8524,E2 445.8503} C_DIS
LIN {X 141.3069,Y 14.3982,Z 189,A 9.5437,B 1.6903,C 0.0966,E1 1.852,E2 444.2577} C_DIS
LIN {X 140.8751,Y 18.1288,Z 189,A 10.7916,B 1.6905,C 0.0943,E1 1.8516,E2 443.0447} C_DIS
LIN {X 140.4802,Y 20.9813,Z 189,A 12.028,B 1.6907,C 0.0905,E1 1.8511,E2 441.7978} C_DIS
LIN {X 139.7628,Y 25.3134,Z 189,A 13.6556,B 1.6909,C 0.0866,E1 1.8503,E2 440.1883} C_DIS
LIN {X 138.5808,Y 31.1434,Z 189,A 15.8328,B 1.6911,C 0.0816,E1 1.8491,E2 438.0396} C_DIS
LIN {X 137.7198,Y 34.7503,Z 189,A 17.1867,B 1.6913,C 0.0785,E1 1.8482,E2 436.7038} C_DIS
LIN {X 136.5871,Y 38.9716,Z 189,A 19.0787,B 1.6915,C 0.0728,E1 1.8468,E2 434.794} C_DIS
LIN {X 135.62,Y 42.213,Z 189,A 20.1567,B 1.6915,C 0.0711,E1 1.8459,E2 433.7533} C_DIS
LIN {X 134.2717,Y 46.3186,Z 189,A 21.6619,B 1.6917,C 0.0681,E1 1.8446,E2 432.2787} C_DIS
LIN {X 133.0982,Y 49.59,Z 189,A 22.9987,B 1.6918,C 0.0648,E1 1.8433,E2 430.9498} C_DIS
LIN {X 131.7429,Y 53.0854,Z 189,A 24.3293,B 1.6919,C 0.0621,E1 1.842,E2 429.6424} C_DIS
LIN {X 130.5825,Y 55.8812,Z 189,A 25.4482,B 1.692,C 0.0596,E1 1.8408,E2 428.5365} C_DIS
LIN {X 129.1063,Y 59.2114,Z 189,A 26.9132,B 1.6922,C 0.0558,E1 1.8391,E2 427.0714} C_DIS
LIN {X 127.7177,Y 62.1529,Z 189,A 28.1382,B 1.6922,C 0.053,E1 1.8376,E2 425.8574} C_DIS
LIN {X 126.1233,Y 65.3281,Z 189,A 29.5489,B 1.6924,C 0.0495,E1 1.8358,E2 424.4493} C_DIS
LIN {X 123.9812,Y 69.3078,Z 189,A 31.2494,B 1.6924,C 0.0457,E1 1.8336,E2 422.7641} C_DIS
LIN {X 121.6022,Y 73.4011,Z 189,A 32.9755,B 1.6926,C 0.0422,E1 1.8311,E2 421.0613} C_DIS
LIN {X 119.7354,Y 76.4087,Z 189,A 34.3722,B 1.6926,C 0.0389,E1 1.8291,E2 419.6682} C_DIS
LIN {X 117.0364,Y 80.4816,Z 189,A 36.1299,B 1.6927,C 0.0356,E1 1.8264,E2 417.9376} C_DIS
LIN {X 114.5926,Y 83.9248,Z 189,A 37.7686,B 1.6927,C 0.032,E1 1.8237,E2 416.3068} C_DIS
LIN {X 111.7312,Y 87.698,Z 189,A 39.513,B 1.6928,C 0.0287,E1 1.8207,E2 414.5833} C_DIS
LIN {X 109.1539,Y 90.8866,Z 189,A 41.0563,B 1.6928,C 0.0256,E1 1.818,E2 413.0538} C_DIS
Enddeposition()
END
